   1:  PR[GP1:91,1] = PR[GP1:90,1] + -0.626;
   1:  PR[GP1:91,2] = PR[GP1:90,2] + -44.019;
   1:L PR[91] R[100]mm/sec CNT100;
   1:  PR[GP1:91,1] = PR[GP1:90,1] + 0.841;
   1:L PR[91] R[100]mm/sec CNT100;
   1:  PR[GP1:91,1] = PR[GP1:90,1] + 8.391;
   1:  PR[GP1:91,2] = PR[GP1:90,2] + -44.216;
   1:L PR[91] R[100]mm/sec CNT100;
   1:  PR[GP1:91,1] = PR[GP1:90,1] + 12.992;
   1:  PR[GP1:91,2] = PR[GP1:90,2] + -44.314;
   1:L PR[91] R[100]mm/sec CNT100;
   1:  PR[GP1:91,1] = PR[GP1:90,1] + 15.543;
   1:  PR[GP1:91,2] = PR[GP1:90,2] + -43.998;
   1:L PR[91] R[100]mm/sec CNT100;
   1:  PR[GP1:91,1] = PR[GP1:90,1] + 27.793;
   1:  PR[GP1:91,2] = PR[GP1:90,2] + -39.874;
   1:L PR[91] R[100]mm/sec CNT100;
   1:  PR[GP1:91,1] = PR[GP1:90,1] + 29.749;
   1:  PR[GP1:91,2] = PR[GP1:90,2] + -39.116;
   1:L PR[91] R[100]mm/sec CNT100;
   1:  PR[GP1:91,1] = PR[GP1:90,1] + 40.362;
   1:  PR[GP1:91,2] = PR[GP1:90,2] + -30.633;
   1:L PR[91] R[100]mm/sec CNT100;
   1:  PR[GP1:91,1] = PR[GP1:90,1] + 41.764;
   1:  PR[GP1:91,2] = PR[GP1:90,2] + -29.640;
   1:L PR[91] R[100]mm/sec CNT100;
   1:  PR[GP1:91,1] = PR[GP1:90,1] + 42.961;
   1:  PR[GP1:91,2] = PR[GP1:90,2] + -28.198;
   1:L PR[91] R[100]mm/sec CNT100;
   1:  PR[GP1:91,1] = PR[GP1:90,1] + 49.960;
   1:  PR[GP1:91,2] = PR[GP1:90,2] + -16.511;
   1:L PR[91] R[100]mm/sec CNT100;
   1:  PR[GP1:91,1] = PR[GP1:90,1] + 50.589;
   1:  PR[GP1:91,2] = PR[GP1:90,2] + -15.086;
   1:L PR[91] R[100]mm/sec CNT100;
   1:  PR[GP1:91,1] = PR[GP1:90,1] + 53.075;
   1:  PR[GP1:91,2] = PR[GP1:90,2] + -1.444;
   1:L PR[91] R[100]mm/sec CNT100;
   1:  PR[GP1:91,1] = PR[GP1:90,1] + 53.265;
   1:  PR[GP1:91,2] = PR[GP1:90,2] + -0.085;
   1:L PR[91] R[100]mm/sec CNT100;
   1:  PR[GP1:91,1] = PR[GP1:90,1] + 50.804;
   1:  PR[GP1:91,2] = PR[GP1:90,2] + 13.373;
   1:L PR[91] R[100]mm/sec CNT100;
   1:  PR[GP1:91,1] = PR[GP1:90,1] + 50.584;
   1:  PR[GP1:91,2] = PR[GP1:90,2] + 14.954;
   1:L PR[91] R[100]mm/sec CNT100;
   1:  PR[GP1:91,1] = PR[GP1:90,1] + 49.959;
   1:  PR[GP1:91,2] = PR[GP1:90,2] + 16.368;
   1:L PR[91] R[100]mm/sec CNT100;
   1:  PR[GP1:91,1] = PR[GP1:90,1] + 42.960;
   1:  PR[GP1:91,2] = PR[GP1:90,2] + 28.055;
   1:L PR[91] R[100]mm/sec CNT100;
   1:  PR[GP1:91,1] = PR[GP1:90,1] + 41.751;
   1:  PR[GP1:91,2] = PR[GP1:90,2] + 29.511;
   1:L PR[91] R[100]mm/sec CNT100;
   1:  PR[GP1:91,1] = PR[GP1:90,1] + 31.485;
   1:  PR[GP1:91,2] = PR[GP1:90,2] + 37.748;
   1:L PR[91] R[100]mm/sec CNT100;
   1:  PR[GP1:91,1] = PR[GP1:90,1] + 29.763;
   1:  PR[GP1:91,2] = PR[GP1:90,2] + 38.967;
   1:L PR[91] R[100]mm/sec CNT100;
   1:  PR[GP1:91,1] = PR[GP1:90,1] + 27.791;
   1:  PR[GP1:91,2] = PR[GP1:90,2] + 39.731;
   1:L PR[91] R[100]mm/sec CNT100;
   1:  PR[GP1:91,1] = PR[GP1:90,1] + 15.540;
   1:  PR[GP1:91,2] = PR[GP1:90,2] + 43.855;
   1:L PR[91] R[100]mm/sec CNT100;
   1:  PR[GP1:91,1] = PR[GP1:90,1] + 12.988;
   1:  PR[GP1:91,2] = PR[GP1:90,2] + 44.171;
   1:L PR[91] R[100]mm/sec CNT100;
   1:  PR[GP1:91,1] = PR[GP1:90,1] + 8.403;
   1:  PR[GP1:91,2] = PR[GP1:90,2] + 44.072;
   1:L PR[91] R[100]mm/sec CNT100;
   1:  PR[GP1:91,1] = PR[GP1:90,1] + 0.841;
   1:  PR[GP1:91,2] = PR[GP1:90,2] + 43.875;
   1:L PR[91] R[100]mm/sec CNT100;
   1:  ! -- Layer/Ebene 176 -- !;
   1:  PR[91] = PR[90];
   1:  PR[GP1:91,1] = PR[GP1:90,1] + -0.604;
   1:  PR[GP1:91,2] = PR[GP1:90,2] + 44.034;
   1:  PR[GP1:91,3] = PR[GP1:90,3] + 107.665;
   1:L PR[91] R[100]mm/sec CNT100;
   1:  PR[GP1:91,1] = PR[GP1:90,1] + -7.340;
   1:  PR[GP1:91,2] = PR[GP1:90,2] + 44.210;
   1:L PR[91] R[100]mm/sec CNT100;
   1:  PR[GP1:91,1] = PR[GP1:90,1] + -12.403;
   1:  PR[GP1:91,2] = PR[GP1:90,2] + 44.319;
   1:L PR[91] R[100]mm/sec CNT100;
   1:  PR[GP1:91,1] = PR[GP1:90,1] + -15.228;
   1:  PR[GP1:91,2] = PR[GP1:90,2] + 43.969;
   1:L PR[91] R[100]mm/sec CNT100;
   1:  PR[GP1:91,1] = PR[GP1:90,1] + -27.126;
   1:  PR[GP1:91,2] = PR[GP1:90,2] + 39.965;
   1:L PR[91] R[100]mm/sec CNT100;
   1:  PR[GP1:91,1] = PR[GP1:90,1] + -29.351;
   1:  PR[GP1:91,2] = PR[GP1:90,2] + 39.103;
   1:L PR[91] R[100]mm/sec CNT100;
   1:  PR[GP1:91,1] = PR[GP1:90,1] + -39.660;
   1:  PR[GP1:91,2] = PR[GP1:90,2] + 30.866;
   1:L PR[91] R[100]mm/sec CNT100;
   1:  PR[GP1:91,1] = PR[GP1:90,1] + -41.308;
   1:  PR[GP1:91,2] = PR[GP1:90,2] + 29.699;
   1:L PR[91] R[100]mm/sec CNT100;
   1:  PR[GP1:91,1] = PR[GP1:90,1] + -42.722;
   1:  PR[GP1:91,2] = PR[GP1:90,2] + 27.996;
   1:L PR[91] R[100]mm/sec CNT100;
   1:  PR[GP1:91,1] = PR[GP1:90,1] + -49.520;
   1:  PR[GP1:91,2] = PR[GP1:90,2] + 16.640;
   1:L PR[91] R[100]mm/sec CNT100;
   1:  PR[GP1:91,1] = PR[GP1:90,1] + -50.290;
   1:  PR[GP1:91,2] = PR[GP1:90,2] + 14.895;
   1:L PR[91] R[100]mm/sec CNT100;
   1:  PR[GP1:91,1] = PR[GP1:90,1] + -52.705;
   1:  PR[GP1:91,2] = PR[GP1:90,2] + 1.651;
   1:L PR[91] R[100]mm/sec CNT100;
   1:  PR[GP1:91,1] = PR[GP1:90,1] + -52.943;
   1:  PR[GP1:91,2] = PR[GP1:90,2] + -0.059;
   1:L PR[91] R[100]mm/sec CNT100;
   1:  PR[GP1:91,1] = PR[GP1:90,1] + -50.554;
   1:  PR[GP1:91,2] = PR[GP1:90,2] + -13.124;
   1:L PR[91] R[100]mm/sec CNT100;
   1:  PR[GP1:91,1] = PR[GP1:90,1] + -50.285;
   1:  PR[GP1:91,2] = PR[GP1:90,2] + -15.050;
   1:L PR[91] R[100]mm/sec CNT100;
   1:  PR[GP1:91,1] = PR[GP1:90,1] + -49.520;
   1:  PR[GP1:91,2] = PR[GP1:90,2] + -16.783;
   1:L PR[91] R[100]mm/sec CNT100;
   1:  PR[GP1:91,1] = PR[GP1:90,1] + -42.723;
   1:  PR[GP1:91,2] = PR[GP1:90,2] + -28.138;
   1:L PR[91] R[100]mm/sec CNT100;
   1:  PR[GP1:91,1] = PR[GP1:90,1] + -41.297;
   1:  PR[GP1:91,2] = PR[GP1:90,2] + -29.856;
   1:L PR[91] R[100]mm/sec CNT100;
   1:  PR[GP1:91,1] = PR[GP1:90,1] + -31.328;
   1:  PR[GP1:91,2] = PR[GP1:90,2] + -37.852;
   1:L PR[91] R[100]mm/sec CNT100;
   1:  PR[GP1:91,1] = PR[GP1:90,1] + -29.370;
   1:  PR[GP1:91,2] = PR[GP1:90,2] + -39.239;
   1:L PR[91] R[100]mm/sec CNT100;
   1:  PR[GP1:91,1] = PR[GP1:90,1] + -27.129;
   1:  PR[GP1:91,2] = PR[GP1:90,2] + -40.108;
   1:L PR[91] R[100]mm/sec CNT100;
   1:  PR[GP1:91,1] = PR[GP1:90,1] + -15.231;
   1:  PR[GP1:91,2] = PR[GP1:90,2] + -44.113;
   1:L PR[91] R[100]mm/sec CNT100;
   1:  PR[GP1:91,1] = PR[GP1:90,1] + -12.406;
   1:  PR[GP1:91,2] = PR[GP1:90,2] + -44.463;
   1:L PR[91] R[100]mm/sec CNT100;
   1:  PR[GP1:91,1] = PR[GP1:90,1] + -7.326;
   1:  PR[GP1:91,2] = PR[GP1:90,2] + -44.353;
   1:L PR[91] R[100]mm/sec CNT100;
   1:  PR[GP1:91,1] = PR[GP1:90,1] + -0.604;
   1:  PR[GP1:91,2] = PR[GP1:90,2] + -44.178;
   1:L PR[91] R[100]mm/sec CNT100;
   1:  PR[GP1:91,1] = PR[GP1:90,1] + 0.818;
   1:L PR[91] R[100]mm/sec CNT100;
   1:  PR[GP1:91,1] = PR[GP1:90,1] + 7.540;
   1:  PR[GP1:91,2] = PR[GP1:90,2] + -44.353;
   1:L PR[91] R[100]mm/sec CNT100;
   1:  PR[GP1:91,1] = PR[GP1:90,1] + 12.621;
   1:  PR[GP1:91,2] = PR[GP1:90,2] + -44.462;
   1:L PR[91] R[100]mm/sec CNT100;
   1:  PR[GP1:91,1] = PR[GP1:90,1] + 15.446;
   1:  PR[GP1:91,2] = PR[GP1:90,2] + -44.113;
   1:L PR[91] R[100]mm/sec CNT100;
   1:  PR[GP1:91,1] = PR[GP1:90,1] + 27.343;
   1:  PR[GP1:91,2] = PR[GP1:90,2] + -40.107;
   1:L PR[91] R[100]mm/sec CNT100;
   1:  PR[GP1:91,1] = PR[GP1:90,1] + 29.568;
   1:  PR[GP1:91,2] = PR[GP1:90,2] + -39.245;
   1:L PR[91] R[100]mm/sec CNT100;
   1:  PR[GP1:91,1] = PR[GP1:90,1] + 39.875;
   1:  PR[GP1:91,2] = PR[GP1:90,2] + -31.006;
   1:L PR[91] R[100]mm/sec CNT100;
   1:  PR[GP1:91,1] = PR[GP1:90,1] + 41.523;
   1:  PR[GP1:91,2] = PR[GP1:90,2] + -29.839;
   1:L PR[91] R[100]mm/sec CNT100;
   1:  PR[GP1:91,1] = PR[GP1:90,1] + 42.937;
   1:  PR[GP1:91,2] = PR[GP1:90,2] + -28.136;
   1:L PR[91] R[100]mm/sec CNT100;
   1:  PR[GP1:91,1] = PR[GP1:90,1] + 49.733;
   1:  PR[GP1:91,2] = PR[GP1:90,2] + -16.787;
   1:L PR[91] R[100]mm/sec CNT100;
   1:  PR[GP1:91,1] = PR[GP1:90,1] + 50.504;
   1:  PR[GP1:91,2] = PR[GP1:90,2] + -15.042;
   1:L PR[91] R[100]mm/sec CNT100;
   1:  PR[GP1:91,1] = PR[GP1:90,1] + 52.918;
   1:  PR[GP1:91,2] = PR[GP1:90,2] + -1.795;
   1:L PR[91] R[100]mm/sec CNT100;
   1:  PR[GP1:91,1] = PR[GP1:90,1] + 53.157;
   1:  PR[GP1:91,2] = PR[GP1:90,2] + -0.085;
   1:L PR[91] R[100]mm/sec CNT100;
   1:  PR[GP1:91,1] = PR[GP1:90,1] + 50.767;
   1:  PR[GP1:91,2] = PR[GP1:90,2] + 12.985;
   1:L PR[91] R[100]mm/sec CNT100;
   1:  PR[GP1:91,1] = PR[GP1:90,1] + 50.498;
   1:  PR[GP1:91,2] = PR[GP1:90,2] + 14.911;
   1:L PR[91] R[100]mm/sec CNT100;
   1:  PR[GP1:91,1] = PR[GP1:90,1] + 49.733;
   1:  PR[GP1:91,2] = PR[GP1:90,2] + 16.644;
   1:L PR[91] R[100]mm/sec CNT100;
   1:  PR[GP1:91,1] = PR[GP1:90,1] + 42.936;
   1:  PR[GP1:91,2] = PR[GP1:90,2] + 27.993;
   1:L PR[91] R[100]mm/sec CNT100;
   1:  PR[GP1:91,1] = PR[GP1:90,1] + 41.511;
   1:  PR[GP1:91,2] = PR[GP1:90,2] + 29.710;
   1:L PR[91] R[100]mm/sec CNT100;
   1:  PR[GP1:91,1] = PR[GP1:90,1] + 31.541;
   1:  PR[GP1:91,2] = PR[GP1:90,2] + 37.709;
   1:L PR[91] R[100]mm/sec CNT100;
   1:  PR[GP1:91,1] = PR[GP1:90,1] + 29.583;
   1:  PR[GP1:91,2] = PR[GP1:90,2] + 39.096;
   1:L PR[91] R[100]mm/sec CNT100;
   1:  PR[GP1:91,1] = PR[GP1:90,1] + 27.341;
   1:  PR[GP1:91,2] = PR[GP1:90,2] + 39.964;
   1:L PR[91] R[100]mm/sec CNT100;
   1:  PR[GP1:91,1] = PR[GP1:90,1] + 15.443;
   1:  PR[GP1:91,2] = PR[GP1:90,2] + 43.969;
   1:L PR[91] R[100]mm/sec CNT100;
   1:  PR[GP1:91,1] = PR[GP1:90,1] + 12.618;
   1:  PR[GP1:91,2] = PR[GP1:90,2] + 44.319;
   1:L PR[91] R[100]mm/sec CNT100;
   1:  PR[GP1:91,1] = PR[GP1:90,1] + 7.554;
   1:  PR[GP1:91,2] = PR[GP1:90,2] + 44.210;
   1:L PR[91] R[100]mm/sec CNT100;
   1:  PR[GP1:91,1] = PR[GP1:90,1] + 0.818;
   1:  PR[GP1:91,2] = PR[GP1:90,2] + 44.034;
   1:L PR[91] R[100]mm/sec CNT100;
   1:  ! -- Layer/Ebene 177 -- !;
   1:  PR[91] = PR[90];
   1:  PR[GP1:91,1] = PR[GP1:90,1] + -0.581;
   1:  PR[GP1:91,2] = PR[GP1:90,2] + 44.194;
   1:  PR[GP1:91,3] = PR[GP1:90,3] + 108.275;
   1:L PR[91] R[100]mm/sec CNT100;
   1:  PR[GP1:91,1] = PR[GP1:90,1] + -6.491;
   1:  PR[GP1:91,2] = PR[GP1:90,2] + 44.348;
   1:L PR[91] R[100]mm/sec CNT100;
   1:  PR[GP1:91,1] = PR[GP1:90,1] + -12.033;
   1:  PR[GP1:91,2] = PR[GP1:90,2] + 44.467;
   1:L PR[91] R[100]mm/sec CNT100;
   1:  PR[GP1:91,1] = PR[GP1:90,1] + -15.132;
   1:  PR[GP1:91,2] = PR[GP1:90,2] + 44.083;
   1:L PR[91] R[100]mm/sec CNT100;
   1:  PR[GP1:91,1] = PR[GP1:90,1] + -26.676;
   1:  PR[GP1:91,2] = PR[GP1:90,2] + 40.198;
   1:L PR[91] R[100]mm/sec CNT100;
   1:  PR[GP1:91,1] = PR[GP1:90,1] + -29.171;
   1:  PR[GP1:91,2] = PR[GP1:90,2] + 39.231;
   1:L PR[91] R[100]mm/sec CNT100;
   1:  PR[GP1:91,1] = PR[GP1:90,1] + -39.173;
   1:  PR[GP1:91,2] = PR[GP1:90,2] + 31.240;
   1:L PR[91] R[100]mm/sec CNT100;
   1:  PR[GP1:91,1] = PR[GP1:90,1] + -41.068;
   1:  PR[GP1:91,2] = PR[GP1:90,2] + 29.898;
   1:L PR[91] R[100]mm/sec CNT100;
   1:  PR[GP1:91,1] = PR[GP1:90,1] + -42.698;
   1:  PR[GP1:91,2] = PR[GP1:90,2] + 27.934;
   1:L PR[91] R[100]mm/sec CNT100;
   1:  PR[GP1:91,1] = PR[GP1:90,1] + -49.294;
   1:  PR[GP1:91,2] = PR[GP1:90,2] + 16.916;
   1:L PR[91] R[100]mm/sec CNT100;
   1:  PR[GP1:91,1] = PR[GP1:90,1] + -50.205;
   1:  PR[GP1:91,2] = PR[GP1:90,2] + 14.852;
   1:L PR[91] R[100]mm/sec CNT100;
   1:  PR[GP1:91,1] = PR[GP1:90,1] + -52.548;
   1:  PR[GP1:91,2] = PR[GP1:90,2] + 2.002;
   1:L PR[91] R[100]mm/sec CNT100;
   1:  PR[GP1:91,1] = PR[GP1:90,1] + -52.835;
   1:  PR[GP1:91,2] = PR[GP1:90,2] + -0.059;
   1:L PR[91] R[100]mm/sec CNT100;
   1:  PR[GP1:91,1] = PR[GP1:90,1] + -50.517;
   1:  PR[GP1:91,2] = PR[GP1:90,2] + -12.735;
   1:L PR[91] R[100]mm/sec CNT100;
   1:  PR[GP1:91,1] = PR[GP1:90,1] + -50.200;
   1:  PR[GP1:91,2] = PR[GP1:90,2] + -15.007;
   1:L PR[91] R[100]mm/sec CNT100;
   1:  PR[GP1:91,1] = PR[GP1:90,1] + -49.294;
   1:  PR[GP1:91,2] = PR[GP1:90,2] + -17.059;
   1:L PR[91] R[100]mm/sec CNT100;
   1:  PR[GP1:91,1] = PR[GP1:90,1] + -42.699;
   1:  PR[GP1:91,2] = PR[GP1:90,2] + -28.076;
   1:L PR[91] R[100]mm/sec CNT100;
   1:  PR[GP1:91,1] = PR[GP1:90,1] + -41.057;
   1:  PR[GP1:91,2] = PR[GP1:90,2] + -30.055;
   1:L PR[91] R[100]mm/sec CNT100;
   1:  PR[GP1:91,1] = PR[GP1:90,1] + -31.384;
   1:  PR[GP1:91,2] = PR[GP1:90,2] + -37.813;
   1:L PR[91] R[100]mm/sec CNT100;
   1:  PR[GP1:91,1] = PR[GP1:90,1] + -29.190;
   1:  PR[GP1:91,2] = PR[GP1:90,2] + -39.367;
   1:L PR[91] R[100]mm/sec CNT100;
   1:  PR[GP1:91,1] = PR[GP1:90,1] + -26.678;
   1:  PR[GP1:91,2] = PR[GP1:90,2] + -40.341;
   1:L PR[91] R[100]mm/sec CNT100;
   1:  PR[GP1:91,1] = PR[GP1:90,1] + -15.135;
   1:  PR[GP1:91,2] = PR[GP1:90,2] + -44.227;
   1:L PR[91] R[100]mm/sec CNT100;
   1:  PR[GP1:91,1] = PR[GP1:90,1] + -12.036;
   1:  PR[GP1:91,2] = PR[GP1:90,2] + -44.611;
   1:L PR[91] R[100]mm/sec CNT100;
   1:  PR[GP1:91,1] = PR[GP1:90,1] + -6.476;
   1:  PR[GP1:91,2] = PR[GP1:90,2] + -44.491;
   1:L PR[91] R[100]mm/sec CNT100;
   1:  PR[GP1:91,1] = PR[GP1:90,1] + -0.581;
   1:  PR[GP1:91,2] = PR[GP1:90,2] + -44.338;
   1:L PR[91] R[100]mm/sec CNT100;
   1:  PR[GP1:91,1] = PR[GP1:90,1] + 0.795;
   1:L PR[91] R[100]mm/sec CNT100;
   1:  PR[GP1:91,1] = PR[GP1:90,1] + 6.690;
   1:  PR[GP1:91,2] = PR[GP1:90,2] + -44.491;
   1:L PR[91] R[100]mm/sec CNT100;
   1:  PR[GP1:91,1] = PR[GP1:90,1] + 12.250;
   1:  PR[GP1:91,2] = PR[GP1:90,2] + -44.610;
   1:L PR[91] R[100]mm/sec CNT100;
   1:  PR[GP1:91,1] = PR[GP1:90,1] + 15.349;
   1:  PR[GP1:91,2] = PR[GP1:90,2] + -44.227;
   1:L PR[91] R[100]mm/sec CNT100;
   1:  PR[GP1:91,1] = PR[GP1:90,1] + 26.893;
   1:  PR[GP1:91,2] = PR[GP1:90,2] + -40.340;
   1:L PR[91] R[100]mm/sec CNT100;
   1:  PR[GP1:91,1] = PR[GP1:90,1] + 29.388;
   1:  PR[GP1:91,2] = PR[GP1:90,2] + -39.373;
   1:L PR[91] R[100]mm/sec CNT100;
   1:  PR[GP1:91,1] = PR[GP1:90,1] + 39.388;
   1:  PR[GP1:91,2] = PR[GP1:90,2] + -31.380;
   1:L PR[91] R[100]mm/sec CNT100;
   1:  PR[GP1:91,1] = PR[GP1:90,1] + 41.283;
   1:  PR[GP1:91,2] = PR[GP1:90,2] + -30.038;
   1:L PR[91] R[100]mm/sec CNT100;
   1:  PR[GP1:91,1] = PR[GP1:90,1] + 42.914;
   1:  PR[GP1:91,2] = PR[GP1:90,2] + -28.074;
   1:L PR[91] R[100]mm/sec CNT100;
   1:  PR[GP1:91,1] = PR[GP1:90,1] + 49.508;
   1:  PR[GP1:91,2] = PR[GP1:90,2] + -17.063;
   1:L PR[91] R[100]mm/sec CNT100;
   1:  PR[GP1:91,1] = PR[GP1:90,1] + 50.419;
   1:  PR[GP1:91,2] = PR[GP1:90,2] + -14.999;
   1:L PR[91] R[100]mm/sec CNT100;
   1:  PR[GP1:91,1] = PR[GP1:90,1] + 52.761;
   1:  PR[GP1:91,2] = PR[GP1:90,2] + -2.146;
   1:L PR[91] R[100]mm/sec CNT100;
   1:  PR[GP1:91,1] = PR[GP1:90,1] + 53.048;
   1:  PR[GP1:91,2] = PR[GP1:90,2] + -0.085;
   1:L PR[91] R[100]mm/sec CNT100;
   1:  PR[GP1:91,1] = PR[GP1:90,1] + 50.730;
   1:  PR[GP1:91,2] = PR[GP1:90,2] + 12.596;
   1:L PR[91] R[100]mm/sec CNT100;
   1:  PR[GP1:91,1] = PR[GP1:90,1] + 50.413;
   1:  PR[GP1:91,2] = PR[GP1:90,2] + 14.867;
   1:L PR[91] R[100]mm/sec CNT100;
   1:  PR[GP1:91,1] = PR[GP1:90,1] + 49.507;
   1:  PR[GP1:91,2] = PR[GP1:90,2] + 16.919;
   1:L PR[91] R[100]mm/sec CNT100;
   1:  PR[GP1:91,1] = PR[GP1:90,1] + 42.912;
   1:  PR[GP1:91,2] = PR[GP1:90,2] + 27.931;
   1:L PR[91] R[100]mm/sec CNT100;
   1:  PR[GP1:91,1] = PR[GP1:90,1] + 41.270;
   1:  PR[GP1:91,2] = PR[GP1:90,2] + 29.909;
   1:L PR[91] R[100]mm/sec CNT100;
   1:  PR[GP1:91,1] = PR[GP1:90,1] + 31.597;
   1:  PR[GP1:91,2] = PR[GP1:90,2] + 37.670;
   1:L PR[91] R[100]mm/sec CNT100;
   1:  PR[GP1:91,1] = PR[GP1:90,1] + 29.402;
   1:  PR[GP1:91,2] = PR[GP1:90,2] + 39.224;
   1:L PR[91] R[100]mm/sec CNT100;
   1:  PR[GP1:91,1] = PR[GP1:90,1] + 26.890;
   1:  PR[GP1:91,2] = PR[GP1:90,2] + 40.198;
   1:L PR[91] R[100]mm/sec CNT100;
   1:  PR[GP1:91,1] = PR[GP1:90,1] + 15.346;
   1:  PR[GP1:91,2] = PR[GP1:90,2] + 44.083;
   1:L PR[91] R[100]mm/sec CNT100;
   1:  PR[GP1:91,1] = PR[GP1:90,1] + 12.247;
   1:  PR[GP1:91,2] = PR[GP1:90,2] + 44.467;
   1:L PR[91] R[100]mm/sec CNT100;
   1:  PR[GP1:91,1] = PR[GP1:90,1] + 6.705;
   1:  PR[GP1:91,2] = PR[GP1:90,2] + 44.348;
   1:L PR[91] R[100]mm/sec CNT100;
   1:  PR[GP1:91,1] = PR[GP1:90,1] + 0.795;
   1:  PR[GP1:91,2] = PR[GP1:90,2] + 44.194;
   1:L PR[91] R[100]mm/sec CNT100;
   1:  ! -- Layer/Ebene 178 -- !;
   1:  PR[91] = PR[90];
   1:  PR[GP1:91,1] = PR[GP1:90,1] + -0.559;
   1:  PR[GP1:91,2] = PR[GP1:90,2] + 44.353;
   1:  PR[GP1:91,3] = PR[GP1:90,3] + 108.885;
   1:L PR[91] R[100]mm/sec CNT100;
   1:  PR[GP1:91,1] = PR[GP1:90,1] + -5.642;
   1:  PR[GP1:91,2] = PR[GP1:90,2] + 44.486;
   1:L PR[91] R[100]mm/sec CNT100;
   1:  PR[GP1:91,1] = PR[GP1:90,1] + -11.662;
   1:  PR[GP1:91,2] = PR[GP1:90,2] + 44.615;
   1:L PR[91] R[100]mm/sec CNT100;
   1:  PR[GP1:91,1] = PR[GP1:90,1] + -15.035;
   1:  PR[GP1:91,2] = PR[GP1:90,2] + 44.197;
   1:L PR[91] R[100]mm/sec CNT100;
   1:  PR[GP1:91,1] = PR[GP1:90,1] + -26.226;
   1:  PR[GP1:91,2] = PR[GP1:90,2] + 40.431;
   1:L PR[91] R[100]mm/sec CNT100;
   1:  PR[GP1:91,1] = PR[GP1:90,1] + -28.991;
   1:  PR[GP1:91,2] = PR[GP1:90,2] + 39.359;
   1:L PR[91] R[100]mm/sec CNT100;
   1:  PR[GP1:91,1] = PR[GP1:90,1] + -38.686;
   1:  PR[GP1:91,2] = PR[GP1:90,2] + 31.613;
   1:L PR[91] R[100]mm/sec CNT100;
   1:  PR[GP1:91,1] = PR[GP1:90,1] + -40.827;
   1:  PR[GP1:91,2] = PR[GP1:90,2] + 30.097;
   1:L PR[91] R[100]mm/sec CNT100;
   1:  PR[GP1:91,1] = PR[GP1:90,1] + -42.675;
   1:  PR[GP1:91,2] = PR[GP1:90,2] + 27.872;
   1:L PR[91] R[100]mm/sec CNT100;
   1:  PR[GP1:91,1] = PR[GP1:90,1] + -49.068;
   1:  PR[GP1:91,2] = PR[GP1:90,2] + 17.191;
   1:L PR[91] R[100]mm/sec CNT100;
   1:  PR[GP1:91,1] = PR[GP1:90,1] + -50.120;
   1:  PR[GP1:91,2] = PR[GP1:90,2] + 14.809;
   1:L PR[91] R[100]mm/sec CNT100;
   1:  PR[GP1:91,1] = PR[GP1:90,1] + -52.391;
   1:  PR[GP1:91,2] = PR[GP1:90,2] + 2.352;
   1:L PR[91] R[100]mm/sec CNT100;
   1:  PR[GP1:91,1] = PR[GP1:90,1] + -52.727;
   1:  PR[GP1:91,2] = PR[GP1:90,2] + -0.059;
   1:L PR[91] R[100]mm/sec CNT100;
   1:  PR[GP1:91,1] = PR[GP1:90,1] + -50.480;
   1:  PR[GP1:91,2] = PR[GP1:90,2] + -12.347;
   1:L PR[91] R[100]mm/sec CNT100;
   1:  PR[GP1:91,1] = PR[GP1:90,1] + -50.115;
   1:  PR[GP1:91,2] = PR[GP1:90,2] + -14.963;
   1:L PR[91] R[100]mm/sec CNT100;
   1:  PR[GP1:91,1] = PR[GP1:90,1] + -49.068;
   1:  PR[GP1:91,2] = PR[GP1:90,2] + -17.335;
   1:L PR[91] R[100]mm/sec CNT100;
   1:  PR[GP1:91,1] = PR[GP1:90,1] + -42.676;
   1:  PR[GP1:91,2] = PR[GP1:90,2] + -28.014;
   1:L PR[91] R[100]mm/sec CNT100;
   1:  PR[GP1:91,1] = PR[GP1:90,1] + -40.817;
   1:  PR[GP1:91,2] = PR[GP1:90,2] + -30.254;
   1:L PR[91] R[100]mm/sec CNT100;
   1:  PR[GP1:91,1] = PR[GP1:90,1] + -31.440;
   1:  PR[GP1:91,2] = PR[GP1:90,2] + -37.774;
   1:L PR[91] R[100]mm/sec CNT100;
   1:  PR[GP1:91,1] = PR[GP1:90,1] + -29.009;
   1:  PR[GP1:91,2] = PR[GP1:90,2] + -39.496;
   1:L PR[91] R[100]mm/sec CNT100;
   1:  PR[GP1:91,1] = PR[GP1:90,1] + -26.228;
   1:  PR[GP1:91,2] = PR[GP1:90,2] + -40.574;
   1:L PR[91] R[100]mm/sec CNT100;
   1:  PR[GP1:91,1] = PR[GP1:90,1] + -15.038;
   1:  PR[GP1:91,2] = PR[GP1:90,2] + -44.341;
   1:L PR[91] R[100]mm/sec CNT100;
   1:  PR[GP1:91,1] = PR[GP1:90,1] + -11.665;
   1:  PR[GP1:91,2] = PR[GP1:90,2] + -44.759;
   1:L PR[91] R[100]mm/sec CNT100;
   1:  PR[GP1:91,1] = PR[GP1:90,1] + -5.625;
   1:  PR[GP1:91,2] = PR[GP1:90,2] + -44.629;
   1:L PR[91] R[100]mm/sec CNT100;
   1:  PR[GP1:91,1] = PR[GP1:90,1] + -0.559;
   1:  PR[GP1:91,2] = PR[GP1:90,2] + -44.497;
   1:L PR[91] R[100]mm/sec CNT100;
   1:  PR[GP1:91,1] = PR[GP1:90,1] + 0.772;
   1:L PR[91] R[100]mm/sec CNT100;
   1:  PR[GP1:91,1] = PR[GP1:90,1] + 5.839;
   1:  PR[GP1:91,2] = PR[GP1:90,2] + -44.629;
   1:L PR[91] R[100]mm/sec CNT100;
   1:  PR[GP1:91,1] = PR[GP1:90,1] + 11.879;
   1:  PR[GP1:91,2] = PR[GP1:90,2] + -44.759;
   1:L PR[91] R[100]mm/sec CNT100;
   1:  PR[GP1:91,1] = PR[GP1:90,1] + 15.252;
   1:  PR[GP1:91,2] = PR[GP1:90,2] + -44.341;
   1:L PR[91] R[100]mm/sec CNT100;
   1:  PR[GP1:91,1] = PR[GP1:90,1] + 26.442;
   1:  PR[GP1:91,2] = PR[GP1:90,2] + -40.573;
   1:L PR[91] R[100]mm/sec CNT100;
   1:  PR[GP1:91,1] = PR[GP1:90,1] + 29.207;
   1:  PR[GP1:91,2] = PR[GP1:90,2] + -39.502;
   1:L PR[91] R[100]mm/sec CNT100;
   1:  PR[GP1:91,1] = PR[GP1:90,1] + 38.901;
   1:  PR[GP1:91,2] = PR[GP1:90,2] + -31.753;
   1:L PR[91] R[100]mm/sec CNT100;
   1:  PR[GP1:91,1] = PR[GP1:90,1] + 41.043;
   1:  PR[GP1:91,2] = PR[GP1:90,2] + -30.237;
   1:L PR[91] R[100]mm/sec CNT100;
   1:  PR[GP1:91,1] = PR[GP1:90,1] + 42.890;
   1:  PR[GP1:91,2] = PR[GP1:90,2] + -28.012;
   1:L PR[91] R[100]mm/sec CNT100;
   1:  PR[GP1:91,1] = PR[GP1:90,1] + 49.282;
   1:  PR[GP1:91,2] = PR[GP1:90,2] + -17.338;
   1:L PR[91] R[100]mm/sec CNT100;
   1:  PR[GP1:91,1] = PR[GP1:90,1] + 50.333;
   1:  PR[GP1:91,2] = PR[GP1:90,2] + -14.956;
   1:L PR[91] R[100]mm/sec CNT100;
   1:  PR[GP1:91,1] = PR[GP1:90,1] + 52.604;
   1:  PR[GP1:91,2] = PR[GP1:90,2] + -2.496;
   1:L PR[91] R[100]mm/sec CNT100;
   1:  PR[GP1:91,1] = PR[GP1:90,1] + 52.940;
   1:  PR[GP1:91,2] = PR[GP1:90,2] + -0.085;
   1:L PR[91] R[100]mm/sec CNT100;
   1:  PR[GP1:91,1] = PR[GP1:90,1] + 50.693;
   1:  PR[GP1:91,2] = PR[GP1:90,2] + 12.207;
   1:L PR[91] R[100]mm/sec CNT100;
   1:  PR[GP1:91,1] = PR[GP1:90,1] + 50.328;
   1:  PR[GP1:91,2] = PR[GP1:90,2] + 14.824;
   1:L PR[91] R[100]mm/sec CNT100;
   1:  PR[GP1:91,1] = PR[GP1:90,1] + 49.281;
   1:  PR[GP1:91,2] = PR[GP1:90,2] + 17.195;
   1:L PR[91] R[100]mm/sec CNT100;
   1:  PR[GP1:91,1] = PR[GP1:90,1] + 42.889;
   1:  PR[GP1:91,2] = PR[GP1:90,2] + 27.869;
   1:L PR[91] R[100]mm/sec CNT100;
   1:  PR[GP1:91,1] = PR[GP1:90,1] + 41.030;
   1:  PR[GP1:91,2] = PR[GP1:90,2] + 30.108;
   1:L PR[91] R[100]mm/sec CNT100;
   1:  PR[GP1:91,1] = PR[GP1:90,1] + 31.653;
   1:  PR[GP1:91,2] = PR[GP1:90,2] + 37.631;
   1:L PR[91] R[100]mm/sec CNT100;
   1:  PR[GP1:91,1] = PR[GP1:90,1] + 29.222;
   1:  PR[GP1:91,2] = PR[GP1:90,2] + 39.353;
   1:L PR[91] R[100]mm/sec CNT100;
   1:  PR[GP1:91,1] = PR[GP1:90,1] + 26.440;
   1:  PR[GP1:91,2] = PR[GP1:90,2] + 40.431;
   1:L PR[91] R[100]mm/sec CNT100;
   1:  PR[GP1:91,1] = PR[GP1:90,1] + 15.250;
   1:  PR[GP1:91,2] = PR[GP1:90,2] + 44.197;
   1:L PR[91] R[100]mm/sec CNT100;
   1:  PR[GP1:91,1] = PR[GP1:90,1] + 11.876;
   1:  PR[GP1:91,2] = PR[GP1:90,2] + 44.615;
   1:L PR[91] R[100]mm/sec CNT100;
   1:  PR[GP1:91,1] = PR[GP1:90,1] + 5.857;
   1:  PR[GP1:91,2] = PR[GP1:90,2] + 44.485;
   1:L PR[91] R[100]mm/sec CNT100;
   1:  PR[GP1:91,1] = PR[GP1:90,1] + 0.772;
   1:  PR[GP1:91,2] = PR[GP1:90,2] + 44.353;
   1:L PR[91] R[100]mm/sec CNT100;
   1:  ! -- Layer/Ebene 179 -- !;
   1:  PR[91] = PR[90];
   1:  PR[GP1:91,1] = PR[GP1:90,1] + -0.536;
   1:  PR[GP1:91,2] = PR[GP1:90,2] + 44.512;
   1:  PR[GP1:91,3] = PR[GP1:90,3] + 109.495;
   1:L PR[91] R[100]mm/sec CNT100;
   1:  PR[GP1:91,1] = PR[GP1:90,1] + -4.794;
   1:  PR[GP1:91,2] = PR[GP1:90,2] + 44.623;
   1:L PR[91] R[100]mm/sec CNT100;
   1:  PR[GP1:91,1] = PR[GP1:90,1] + -11.291;
   1:  PR[GP1:91,2] = PR[GP1:90,2] + 44.763;
   1:L PR[91] R[100]mm/sec CNT100;
   1:  PR[GP1:91,1] = PR[GP1:90,1] + -14.938;
   1:  PR[GP1:91,2] = PR[GP1:90,2] + 44.311;
   1:L PR[91] R[100]mm/sec CNT100;
   1:  PR[GP1:91,1] = PR[GP1:90,1] + -25.775;
   1:  PR[GP1:91,2] = PR[GP1:90,2] + 40.664;
   1:L PR[91] R[100]mm/sec CNT100;
   1:  PR[GP1:91,1] = PR[GP1:90,1] + -28.811;
   1:  PR[GP1:91,2] = PR[GP1:90,2] + 39.488;
   1:L PR[91] R[100]mm/sec CNT100;
   1:  PR[GP1:91,1] = PR[GP1:90,1] + -38.200;
   1:  PR[GP1:91,2] = PR[GP1:90,2] + 31.986;
   1:L PR[91] R[100]mm/sec CNT100;
   1:  PR[GP1:91,1] = PR[GP1:90,1] + -40.587;
   1:  PR[GP1:91,2] = PR[GP1:90,2] + 30.296;
   1:L PR[91] R[100]mm/sec CNT100;
   1:  PR[GP1:91,1] = PR[GP1:90,1] + -42.651;
   1:  PR[GP1:91,2] = PR[GP1:90,2] + 27.810;
   1:L PR[91] R[100]mm/sec CNT100;
   1:  PR[GP1:91,1] = PR[GP1:90,1] + -48.842;
   1:  PR[GP1:91,2] = PR[GP1:90,2] + 17.467;
   1:L PR[91] R[100]mm/sec CNT100;
   1:  PR[GP1:91,1] = PR[GP1:90,1] + -50.034;
   1:  PR[GP1:91,2] = PR[GP1:90,2] + 14.765;
   1:L PR[91] R[100]mm/sec CNT100;
   1:  PR[GP1:91,1] = PR[GP1:90,1] + -52.234;
   1:  PR[GP1:91,2] = PR[GP1:90,2] + 2.703;
   1:L PR[91] R[100]mm/sec CNT100;
   1:  PR[GP1:91,1] = PR[GP1:90,1] + -52.619;
   1:  PR[GP1:91,2] = PR[GP1:90,2] + -0.059;
   1:L PR[91] R[100]mm/sec CNT100;
   1:  PR[GP1:91,1] = PR[GP1:90,1] + -50.443;
   1:  PR[GP1:91,2] = PR[GP1:90,2] + -11.958;
   1:L PR[91] R[100]mm/sec CNT100;
   1:  PR[GP1:91,1] = PR[GP1:90,1] + -50.030;
   1:  PR[GP1:91,2] = PR[GP1:90,2] + -14.920;
   1:L PR[91] R[100]mm/sec CNT100;
   1:  PR[GP1:91,1] = PR[GP1:90,1] + -48.842;
   1:  PR[GP1:91,2] = PR[GP1:90,2] + -17.610;
   1:L PR[91] R[100]mm/sec CNT100;
   1:  PR[GP1:91,1] = PR[GP1:90,1] + -42.652;
   1:  PR[GP1:91,2] = PR[GP1:90,2] + -27.953;
   1:L PR[91] R[100]mm/sec CNT100;
   1:  PR[GP1:91,1] = PR[GP1:90,1] + -40.576;
   1:  PR[GP1:91,2] = PR[GP1:90,2] + -30.453;
   1:L PR[91] R[100]mm/sec CNT100;
   1:  PR[GP1:91,1] = PR[GP1:90,1] + -31.496;
   1:  PR[GP1:91,2] = PR[GP1:90,2] + -37.736;
   1:L PR[91] R[100]mm/sec CNT100;
   1:  PR[GP1:91,1] = PR[GP1:90,1] + -28.829;
   1:  PR[GP1:91,2] = PR[GP1:90,2] + -39.624;
   1:L PR[91] R[100]mm/sec CNT100;
   1:  PR[GP1:91,1] = PR[GP1:90,1] + -25.777;
   1:  PR[GP1:91,2] = PR[GP1:90,2] + -40.807;
   1:L PR[91] R[100]mm/sec CNT100;
   1:  PR[GP1:91,1] = PR[GP1:90,1] + -14.941;
   1:  PR[GP1:91,2] = PR[GP1:90,2] + -44.455;
   1:L PR[91] R[100]mm/sec CNT100;
   1:  PR[GP1:91,1] = PR[GP1:90,1] + -11.294;
   1:  PR[GP1:91,2] = PR[GP1:90,2] + -44.907;
   1:L PR[91] R[100]mm/sec CNT100;
   1:  PR[GP1:91,1] = PR[GP1:90,1] + -4.775;
   1:  PR[GP1:91,2] = PR[GP1:90,2] + -44.767;
   1:L PR[91] R[100]mm/sec CNT100;
   1:  PR[GP1:91,1] = PR[GP1:90,1] + -0.536;
   1:  PR[GP1:91,2] = PR[GP1:90,2] + -44.656;
   1:L PR[91] R[100]mm/sec CNT100;
   1:  PR[GP1:91,1] = PR[GP1:90,1] + 0.750;
   1:L PR[91] R[100]mm/sec CNT100;
   1:  PR[GP1:91,1] = PR[GP1:90,1] + 4.989;
   1:  PR[GP1:91,2] = PR[GP1:90,2] + -44.767;
   1:L PR[91] R[100]mm/sec CNT100;
   1:  PR[GP1:91,1] = PR[GP1:90,1] + 11.508;
   1:  PR[GP1:91,2] = PR[GP1:90,2] + -44.907;
   1:L PR[91] R[100]mm/sec CNT100;
   1:  PR[GP1:91,1] = PR[GP1:90,1] + 15.156;
   1:  PR[GP1:91,2] = PR[GP1:90,2] + -44.455;
   1:L PR[91] R[100]mm/sec CNT100;
   1:  PR[GP1:91,1] = PR[GP1:90,1] + 25.992;
   1:  PR[GP1:91,2] = PR[GP1:90,2] + -40.807;
   1:L PR[91] R[100]mm/sec CNT100;
   1:  PR[GP1:91,1] = PR[GP1:90,1] + 29.027;
   1:  PR[GP1:91,2] = PR[GP1:90,2] + -39.631;
   1:L PR[91] R[100]mm/sec CNT100;
   1:  PR[GP1:91,1] = PR[GP1:90,1] + 38.415;
   1:  PR[GP1:91,2] = PR[GP1:90,2] + -32.127;
   1:L PR[91] R[100]mm/sec CNT100;
   1:  PR[GP1:91,1] = PR[GP1:90,1] + 40.802;
   1:  PR[GP1:91,2] = PR[GP1:90,2] + -30.436;
   1:L PR[91] R[100]mm/sec CNT100;
   1:  PR[GP1:91,1] = PR[GP1:90,1] + 42.866;
   1:  PR[GP1:91,2] = PR[GP1:90,2] + -27.950;
   1:L PR[91] R[100]mm/sec CNT100;
   1:  PR[GP1:91,1] = PR[GP1:90,1] + 49.055;
   1:  PR[GP1:91,2] = PR[GP1:90,2] + -17.614;
   1:L PR[91] R[100]mm/sec CNT100;
   1:  PR[GP1:91,1] = PR[GP1:90,1] + 50.248;
   1:  PR[GP1:91,2] = PR[GP1:90,2] + -14.912;
   1:L PR[91] R[100]mm/sec CNT100;
   1:  PR[GP1:91,1] = PR[GP1:90,1] + 52.447;
   1:  PR[GP1:91,2] = PR[GP1:90,2] + -2.847;
   1:L PR[91] R[100]mm/sec CNT100;
   1:  PR[GP1:91,1] = PR[GP1:90,1] + 52.832;
   1:  PR[GP1:91,2] = PR[GP1:90,2] + -0.085;
   1:L PR[91] R[100]mm/sec CNT100;
   1:  PR[GP1:91,1] = PR[GP1:90,1] + 50.656;
   1:  PR[GP1:91,2] = PR[GP1:90,2] + 11.819;
   1:L PR[91] R[100]mm/sec CNT100;
   1:  PR[GP1:91,1] = PR[GP1:90,1] + 50.243;
   1:  PR[GP1:91,2] = PR[GP1:90,2] + 14.781;
   1:L PR[91] R[100]mm/sec CNT100;
   1:  PR[GP1:91,1] = PR[GP1:90,1] + 49.055;
   1:  PR[GP1:91,2] = PR[GP1:90,2] + 17.471;
   1:L PR[91] R[100]mm/sec CNT100;
   1:  PR[GP1:91,1] = PR[GP1:90,1] + 42.865;
   1:  PR[GP1:91,2] = PR[GP1:90,2] + 27.807;
   1:L PR[91] R[100]mm/sec CNT100;
   1:  PR[GP1:91,1] = PR[GP1:90,1] + 40.789;
   1:  PR[GP1:91,2] = PR[GP1:90,2] + 30.307;
   1:L PR[91] R[100]mm/sec CNT100;
   1:  PR[GP1:91,1] = PR[GP1:90,1] + 31.709;
   1:  PR[GP1:91,2] = PR[GP1:90,2] + 37.592;
   1:L PR[91] R[100]mm/sec CNT100;
   1:  PR[GP1:91,1] = PR[GP1:90,1] + 29.042;
   1:  PR[GP1:91,2] = PR[GP1:90,2] + 39.481;
   1:L PR[91] R[100]mm/sec CNT100;
   1:  PR[GP1:91,1] = PR[GP1:90,1] + 25.990;
   1:  PR[GP1:91,2] = PR[GP1:90,2] + 40.664;
   1:L PR[91] R[100]mm/sec CNT100;
   1:  PR[GP1:91,1] = PR[GP1:90,1] + 15.153;
   1:  PR[GP1:91,2] = PR[GP1:90,2] + 44.311;
   1:L PR[91] R[100]mm/sec CNT100;
   1:  PR[GP1:91,1] = PR[GP1:90,1] + 11.505;
   1:  PR[GP1:91,2] = PR[GP1:90,2] + 44.763;
   1:L PR[91] R[100]mm/sec CNT100;
   1:  PR[GP1:91,1] = PR[GP1:90,1] + 5.008;
   1:  PR[GP1:91,2] = PR[GP1:90,2] + 44.623;
   1:L PR[91] R[100]mm/sec CNT100;
   1:  PR[GP1:91,1] = PR[GP1:90,1] + 0.750;
   1:  PR[GP1:91,2] = PR[GP1:90,2] + 44.512;
   1:L PR[91] R[100]mm/sec CNT100;
   1:  ! -- Layer/Ebene 180 -- !;
   1:  PR[91] = PR[90];
   1:  PR[GP1:91,1] = PR[GP1:90,1] + -0.513;
   1:  PR[GP1:91,2] = PR[GP1:90,2] + 44.671;
   1:  PR[GP1:91,3] = PR[GP1:90,3] + 110.105;
   1:L PR[91] R[100]mm/sec CNT100;
   1:  PR[GP1:91,1] = PR[GP1:90,1] + -3.945;
   1:  PR[GP1:91,2] = PR[GP1:90,2] + 44.761;
   1:L PR[91] R[100]mm/sec CNT100;
   1:  PR[GP1:91,1] = PR[GP1:90,1] + -10.921;
   1:  PR[GP1:91,2] = PR[GP1:90,2] + 44.911;
   1:L PR[91] R[100]mm/sec CNT100;
   1:  PR[GP1:91,1] = PR[GP1:90,1] + -14.842;
   1:  PR[GP1:91,2] = PR[GP1:90,2] + 44.425;
   1:L PR[91] R[100]mm/sec CNT100;
   1:  PR[GP1:91,1] = PR[GP1:90,1] + -25.325;
   1:  PR[GP1:91,2] = PR[GP1:90,2] + 40.897;
   1:L PR[91] R[100]mm/sec CNT100;
   1:  PR[GP1:91,1] = PR[GP1:90,1] + -28.630;
   1:  PR[GP1:91,2] = PR[GP1:90,2] + 39.616;
   1:L PR[91] R[100]mm/sec CNT100;
   1:  PR[GP1:91,1] = PR[GP1:90,1] + -37.713;
   1:  PR[GP1:91,2] = PR[GP1:90,2] + 32.359;
   1:L PR[91] R[100]mm/sec CNT100;
   1:  PR[GP1:91,1] = PR[GP1:90,1] + -40.346;
   1:  PR[GP1:91,2] = PR[GP1:90,2] + 30.495;
   1:L PR[91] R[100]mm/sec CNT100;
   1:  PR[GP1:91,1] = PR[GP1:90,1] + -42.627;
   1:  PR[GP1:91,2] = PR[GP1:90,2] + 27.748;
   1:L PR[91] R[100]mm/sec CNT100;
   1:  PR[GP1:91,1] = PR[GP1:90,1] + -48.616;
   1:  PR[GP1:91,2] = PR[GP1:90,2] + 17.743;
   1:L PR[91] R[100]mm/sec CNT100;
   1:  PR[GP1:91,1] = PR[GP1:90,1] + -49.949;
   1:  PR[GP1:91,2] = PR[GP1:90,2] + 14.722;
   1:L PR[91] R[100]mm/sec CNT100;
   1:  PR[GP1:91,1] = PR[GP1:90,1] + -52.077;
   1:  PR[GP1:91,2] = PR[GP1:90,2] + 3.054;
   1:L PR[91] R[100]mm/sec CNT100;
   1:  PR[GP1:91,1] = PR[GP1:90,1] + -52.511;
   1:  PR[GP1:91,2] = PR[GP1:90,2] + -0.059;
   1:L PR[91] R[100]mm/sec CNT100;
   1:  PR[GP1:91,1] = PR[GP1:90,1] + -50.406;
   1:  PR[GP1:91,2] = PR[GP1:90,2] + -11.569;
   1:L PR[91] R[100]mm/sec CNT100;
   1:  PR[GP1:91,1] = PR[GP1:90,1] + -49.944;
   1:  PR[GP1:91,2] = PR[GP1:90,2] + -14.877;
   1:L PR[91] R[100]mm/sec CNT100;
   1:  PR[GP1:91,1] = PR[GP1:90,1] + -48.616;
   1:  PR[GP1:91,2] = PR[GP1:90,2] + -17.886;
   1:L PR[91] R[100]mm/sec CNT100;
   1:  PR[GP1:91,1] = PR[GP1:90,1] + -42.628;
   1:  PR[GP1:91,2] = PR[GP1:90,2] + -27.891;
   1:L PR[91] R[100]mm/sec CNT100;
   1:  PR[GP1:91,1] = PR[GP1:90,1] + -40.336;
   1:  PR[GP1:91,2] = PR[GP1:90,2] + -30.652;
   1:L PR[91] R[100]mm/sec CNT100;
   1:  PR[GP1:91,1] = PR[GP1:90,1] + -31.552;
   1:  PR[GP1:91,2] = PR[GP1:90,2] + -37.697;
   1:L PR[91] R[100]mm/sec CNT100;
   1:  PR[GP1:91,1] = PR[GP1:90,1] + -28.649;
   1:  PR[GP1:91,2] = PR[GP1:90,2] + -39.753;
   1:L PR[91] R[100]mm/sec CNT100;
   1:  PR[GP1:91,1] = PR[GP1:90,1] + -25.327;
   1:  PR[GP1:91,2] = PR[GP1:90,2] + -41.040;
   1:L PR[91] R[100]mm/sec CNT100;
   1:  PR[GP1:91,1] = PR[GP1:90,1] + -14.845;
   1:  PR[GP1:91,2] = PR[GP1:90,2] + -44.569;
   1:L PR[91] R[100]mm/sec CNT100;
   1:  PR[GP1:91,1] = PR[GP1:90,1] + -10.924;
   1:  PR[GP1:91,2] = PR[GP1:90,2] + -45.055;
   1:L PR[91] R[100]mm/sec CNT100;
   1:  PR[GP1:91,1] = PR[GP1:90,1] + -3.925;
   1:  PR[GP1:91,2] = PR[GP1:90,2] + -44.904;
   1:L PR[91] R[100]mm/sec CNT100;
   1:  PR[GP1:91,1] = PR[GP1:90,1] + -0.514;
   1:  PR[GP1:91,2] = PR[GP1:90,2] + -44.816;
   1:L PR[91] R[100]mm/sec CNT100;
   1:  PR[GP1:91,1] = PR[GP1:90,1] + 0.727;
   1:L PR[91] R[100]mm/sec CNT100;
   1:  PR[GP1:91,1] = PR[GP1:90,1] + 4.138;
   1:  PR[GP1:91,2] = PR[GP1:90,2] + -44.904;
   1:L PR[91] R[100]mm/sec CNT100;
   1:  PR[GP1:91,1] = PR[GP1:90,1] + 11.138;
   1:  PR[GP1:91,2] = PR[GP1:90,2] + -45.055;
   1:L PR[91] R[100]mm/sec CNT100;
   1:  PR[GP1:91,1] = PR[GP1:90,1] + 15.059;
   1:  PR[GP1:91,2] = PR[GP1:90,2] + -44.569;
   1:L PR[91] R[100]mm/sec CNT100;
   1:  PR[GP1:91,1] = PR[GP1:90,1] + 25.541;
   1:  PR[GP1:91,2] = PR[GP1:90,2] + -41.040;
   1:L PR[91] R[100]mm/sec CNT100;
   1:  PR[GP1:91,1] = PR[GP1:90,1] + 28.847;
   1:  PR[GP1:91,2] = PR[GP1:90,2] + -39.759;
   1:L PR[91] R[100]mm/sec CNT100;
   1:  PR[GP1:91,1] = PR[GP1:90,1] + 37.928;
   1:  PR[GP1:91,2] = PR[GP1:90,2] + -32.500;
   1:L PR[91] R[100]mm/sec CNT100;
   1:  PR[GP1:91,1] = PR[GP1:90,1] + 40.562;
   1:  PR[GP1:91,2] = PR[GP1:90,2] + -30.635;
   1:L PR[91] R[100]mm/sec CNT100;
   1:  PR[GP1:91,1] = PR[GP1:90,1] + 42.842;
   1:  PR[GP1:91,2] = PR[GP1:90,2] + -27.888;
   1:L PR[91] R[100]mm/sec CNT100;
   1:  PR[GP1:91,1] = PR[GP1:90,1] + 48.829;
   1:  PR[GP1:91,2] = PR[GP1:90,2] + -17.890;
   1:L PR[91] R[100]mm/sec CNT100;
   1:  PR[GP1:91,1] = PR[GP1:90,1] + 50.163;
   1:  PR[GP1:91,2] = PR[GP1:90,2] + -14.869;
   1:L PR[91] R[100]mm/sec CNT100;
   1:  PR[GP1:91,1] = PR[GP1:90,1] + 52.290;
   1:  PR[GP1:91,2] = PR[GP1:90,2] + -3.197;
   1:L PR[91] R[100]mm/sec CNT100;
   1:  PR[GP1:91,1] = PR[GP1:90,1] + 52.724;
   1:  PR[GP1:91,2] = PR[GP1:90,2] + -0.085;
   1:L PR[91] R[100]mm/sec CNT100;
   1:  PR[GP1:91,1] = PR[GP1:90,1] + 50.619;
   1:  PR[GP1:91,2] = PR[GP1:90,2] + 11.430;
   1:L PR[91] R[100]mm/sec CNT100;
   1:  PR[GP1:91,1] = PR[GP1:90,1] + 50.158;
   1:  PR[GP1:91,2] = PR[GP1:90,2] + 14.737;
   1:L PR[91] R[100]mm/sec CNT100;
   1:  PR[GP1:91,1] = PR[GP1:90,1] + 48.829;
   1:  PR[GP1:91,2] = PR[GP1:90,2] + 17.746;
   1:L PR[91] R[100]mm/sec CNT100;
   1:  PR[GP1:91,1] = PR[GP1:90,1] + 42.841;
   1:  PR[GP1:91,2] = PR[GP1:90,2] + 27.745;
   1:L PR[91] R[100]mm/sec CNT100;
   1:  PR[GP1:91,1] = PR[GP1:90,1] + 40.549;
   1:  PR[GP1:91,2] = PR[GP1:90,2] + 30.506;
   1:L PR[91] R[100]mm/sec CNT100;
   1:  PR[GP1:91,1] = PR[GP1:90,1] + 31.765;
   1:  PR[GP1:91,2] = PR[GP1:90,2] + 37.553;
   1:L PR[91] R[100]mm/sec CNT100;
   1:  PR[GP1:91,1] = PR[GP1:90,1] + 28.861;
   1:  PR[GP1:91,2] = PR[GP1:90,2] + 39.610;
   1:L PR[91] R[100]mm/sec CNT100;
   1:  PR[GP1:91,1] = PR[GP1:90,1] + 25.539;
   1:  PR[GP1:91,2] = PR[GP1:90,2] + 40.897;
   1:L PR[91] R[100]mm/sec CNT100;
   1:  PR[GP1:91,1] = PR[GP1:90,1] + 15.056;
   1:  PR[GP1:91,2] = PR[GP1:90,2] + 44.425;
   1:L PR[91] R[100]mm/sec CNT100;
   1:  PR[GP1:91,1] = PR[GP1:90,1] + 11.135;
   1:  PR[GP1:91,2] = PR[GP1:90,2] + 44.911;
   1:L PR[91] R[100]mm/sec CNT100;
   1:  PR[GP1:91,1] = PR[GP1:90,1] + 4.159;
   1:  PR[GP1:91,2] = PR[GP1:90,2] + 44.761;
   1:L PR[91] R[100]mm/sec CNT100;
   1:  PR[GP1:91,1] = PR[GP1:90,1] + 0.727;
   1:  PR[GP1:91,2] = PR[GP1:90,2] + 44.671;
   1:L PR[91] R[100]mm/sec CNT100;
   1:  ! -- Layer/Ebene 181 -- !;
   1:  PR[91] = PR[90];
   1:  PR[GP1:91,1] = PR[GP1:90,1] + -0.490;
   1:  PR[GP1:91,2] = PR[GP1:90,2] + 44.831;
   1:  PR[GP1:91,3] = PR[GP1:90,3] + 110.715;
   1:L PR[91] R[100]mm/sec CNT100;
   1:  PR[GP1:91,1] = PR[GP1:90,1] + -10.551;
   1:  PR[GP1:91,2] = PR[GP1:90,2] + 45.059;
   1:L PR[91] R[100]mm/sec CNT100;
   1:  PR[GP1:91,1] = PR[GP1:90,1] + -14.745;
   1:  PR[GP1:91,2] = PR[GP1:90,2] + 44.539;
   1:L PR[91] R[100]mm/sec CNT100;
   1:  PR[GP1:91,1] = PR[GP1:90,1] + -24.875;
   1:  PR[GP1:91,2] = PR[GP1:90,2] + 41.130;
   1:L PR[91] R[100]mm/sec CNT100;
   1:  PR[GP1:91,1] = PR[GP1:90,1] + -28.450;
   1:  PR[GP1:91,2] = PR[GP1:90,2] + 39.745;
   1:L PR[91] R[100]mm/sec CNT100;
   1:  PR[GP1:91,1] = PR[GP1:90,1] + -37.226;
   1:  PR[GP1:91,2] = PR[GP1:90,2] + 32.733;
   1:L PR[91] R[100]mm/sec CNT100;
   1:  PR[GP1:91,1] = PR[GP1:90,1] + -40.106;
   1:  PR[GP1:91,2] = PR[GP1:90,2] + 30.694;
   1:L PR[91] R[100]mm/sec CNT100;
   1:  PR[GP1:91,1] = PR[GP1:90,1] + -42.603;
   1:  PR[GP1:91,2] = PR[GP1:90,2] + 27.686;
   1:L PR[91] R[100]mm/sec CNT100;
   1:  PR[GP1:91,1] = PR[GP1:90,1] + -48.390;
   1:  PR[GP1:91,2] = PR[GP1:90,2] + 18.019;
   1:L PR[91] R[100]mm/sec CNT100;
   1:  PR[GP1:91,1] = PR[GP1:90,1] + -49.864;
   1:  PR[GP1:91,2] = PR[GP1:90,2] + 14.679;
   1:L PR[91] R[100]mm/sec CNT100;
   1:  PR[GP1:91,1] = PR[GP1:90,1] + -51.920;
   1:  PR[GP1:91,2] = PR[GP1:90,2] + 3.404;
   1:L PR[91] R[100]mm/sec CNT100;
   1:  PR[GP1:91,1] = PR[GP1:90,1] + -52.403;
   1:  PR[GP1:91,2] = PR[GP1:90,2] + -0.059;
   1:L PR[91] R[100]mm/sec CNT100;
   1:  PR[GP1:91,1] = PR[GP1:90,1] + -50.369;
   1:  PR[GP1:91,2] = PR[GP1:90,2] + -11.181;
   1:L PR[91] R[100]mm/sec CNT100;
   1:  PR[GP1:91,1] = PR[GP1:90,1] + -49.859;
   1:  PR[GP1:91,2] = PR[GP1:90,2] + -14.834;
   1:L PR[91] R[100]mm/sec CNT100;
   1:  PR[GP1:91,1] = PR[GP1:90,1] + -48.390;
   1:  PR[GP1:91,2] = PR[GP1:90,2] + -18.162;
   1:L PR[91] R[100]mm/sec CNT100;
   1:  PR[GP1:91,1] = PR[GP1:90,1] + -42.604;
   1:  PR[GP1:91,2] = PR[GP1:90,2] + -27.829;
   1:L PR[91] R[100]mm/sec CNT100;
   1:  PR[GP1:91,1] = PR[GP1:90,1] + -40.095;
   1:  PR[GP1:91,2] = PR[GP1:90,2] + -30.851;
   1:L PR[91] R[100]mm/sec CNT100;
   1:  PR[GP1:91,1] = PR[GP1:90,1] + -31.608;
   1:  PR[GP1:91,2] = PR[GP1:90,2] + -37.658;
   1:L PR[91] R[100]mm/sec CNT100;
   1:  PR[GP1:91,1] = PR[GP1:90,1] + -28.468;
   1:  PR[GP1:91,2] = PR[GP1:90,2] + -39.881;
   1:L PR[91] R[100]mm/sec CNT100;
   1:  PR[GP1:91,1] = PR[GP1:90,1] + -24.877;
   1:  PR[GP1:91,2] = PR[GP1:90,2] + -41.273;
   1:L PR[91] R[100]mm/sec CNT100;
   1:  PR[GP1:91,1] = PR[GP1:90,1] + -14.748;
   1:  PR[GP1:91,2] = PR[GP1:90,2] + -44.683;
   1:L PR[91] R[100]mm/sec CNT100;
   1:  PR[GP1:91,1] = PR[GP1:90,1] + -10.553;
   1:  PR[GP1:91,2] = PR[GP1:90,2] + -45.203;
   1:L PR[91] R[100]mm/sec CNT100;
   1:  PR[GP1:91,1] = PR[GP1:90,1] + -0.490;
   1:  PR[GP1:91,2] = PR[GP1:90,2] + -44.975;
   1:L PR[91] R[100]mm/sec CNT100;
   1:  PR[GP1:91,1] = PR[GP1:90,1] + 0.703;
   1:L PR[91] R[100]mm/sec CNT100;
   1:  PR[GP1:91,1] = PR[GP1:90,1] + 10.767;
   1:  PR[GP1:91,2] = PR[GP1:90,2] + -45.203;
   1:L PR[91] R[100]mm/sec CNT100;
   1:  PR[GP1:91,1] = PR[GP1:90,1] + 14.962;
   1:  PR[GP1:91,2] = PR[GP1:90,2] + -44.683;
   1:L PR[91] R[100]mm/sec CNT100;
   1:  PR[GP1:91,1] = PR[GP1:90,1] + 25.091;
   1:  PR[GP1:91,2] = PR[GP1:90,2] + -41.273;
   1:L PR[91] R[100]mm/sec CNT100;
   1:  PR[GP1:91,1] = PR[GP1:90,1] + 28.666;
   1:  PR[GP1:91,2] = PR[GP1:90,2] + -39.888;
   1:L PR[91] R[100]mm/sec CNT100;
   1:  PR[GP1:91,1] = PR[GP1:90,1] + 37.441;
   1:  PR[GP1:91,2] = PR[GP1:90,2] + -32.873;
   1:L PR[91] R[100]mm/sec CNT100;
   1:  PR[GP1:91,1] = PR[GP1:90,1] + 40.321;
   1:  PR[GP1:91,2] = PR[GP1:90,2] + -30.834;
   1:L PR[91] R[100]mm/sec CNT100;
   1:  PR[GP1:91,1] = PR[GP1:90,1] + 42.818;
   1:  PR[GP1:91,2] = PR[GP1:90,2] + -27.826;
   1:L PR[91] R[100]mm/sec CNT100;
   1:  PR[GP1:91,1] = PR[GP1:90,1] + 48.603;
   1:  PR[GP1:91,2] = PR[GP1:90,2] + -18.165;
   1:L PR[91] R[100]mm/sec CNT100;
   1:  PR[GP1:91,1] = PR[GP1:90,1] + 50.078;
   1:  PR[GP1:91,2] = PR[GP1:90,2] + -14.826;
   1:L PR[91] R[100]mm/sec CNT100;
   1:  PR[GP1:91,1] = PR[GP1:90,1] + 52.133;
   1:  PR[GP1:91,2] = PR[GP1:90,2] + -3.548;
   1:L PR[91] R[100]mm/sec CNT100;
   1:  PR[GP1:91,1] = PR[GP1:90,1] + 52.616;
   1:  PR[GP1:91,2] = PR[GP1:90,2] + -0.085;
   1:L PR[91] R[100]mm/sec CNT100;
   1:  PR[GP1:91,1] = PR[GP1:90,1] + 50.582;
   1:  PR[GP1:91,2] = PR[GP1:90,2] + 11.041;
   1:L PR[91] R[100]mm/sec CNT100;
   1:  PR[GP1:91,1] = PR[GP1:90,1] + 50.072;
   1:  PR[GP1:91,2] = PR[GP1:90,2] + 14.694;
   1:L PR[91] R[100]mm/sec CNT100;
   1:  PR[GP1:91,1] = PR[GP1:90,1] + 48.603;
   1:  PR[GP1:91,2] = PR[GP1:90,2] + 18.022;
   1:L PR[91] R[100]mm/sec CNT100;
   1:  PR[GP1:91,1] = PR[GP1:90,1] + 42.817;
   1:  PR[GP1:91,2] = PR[GP1:90,2] + 27.683;
   1:L PR[91] R[100]mm/sec CNT100;
   1:  PR[GP1:91,1] = PR[GP1:90,1] + 40.309;
   1:  PR[GP1:91,2] = PR[GP1:90,2] + 30.705;
   1:L PR[91] R[100]mm/sec CNT100;
   1:  PR[GP1:91,1] = PR[GP1:90,1] + 31.821;
   1:  PR[GP1:91,2] = PR[GP1:90,2] + 37.514;
   1:L PR[91] R[100]mm/sec CNT100;
   1:  PR[GP1:91,1] = PR[GP1:90,1] + 28.681;
   1:  PR[GP1:91,2] = PR[GP1:90,2] + 39.738;
   1:L PR[91] R[100]mm/sec CNT100;
   1:  PR[GP1:91,1] = PR[GP1:90,1] + 25.089;
   1:  PR[GP1:91,2] = PR[GP1:90,2] + 41.130;
   1:L PR[91] R[100]mm/sec CNT100;
   1:  PR[GP1:91,1] = PR[GP1:90,1] + 14.960;
   1:  PR[GP1:91,2] = PR[GP1:90,2] + 44.539;
   1:L PR[91] R[100]mm/sec CNT100;
   1:  PR[GP1:91,1] = PR[GP1:90,1] + 10.764;
   1:  PR[GP1:91,2] = PR[GP1:90,2] + 45.059;
   1:L PR[91] R[100]mm/sec CNT100;
   1:  PR[GP1:91,1] = PR[GP1:90,1] + 0.703;
   1:  PR[GP1:91,2] = PR[GP1:90,2] + 44.831;
   1:L PR[91] R[100]mm/sec CNT100;
   1:  ! -- Layer/Ebene 182 -- !;
   1:  PR[91] = PR[90];
   1:  PR[GP1:91,1] = PR[GP1:90,1] + -0.467;
   1:  PR[GP1:91,2] = PR[GP1:90,2] + 44.990;
   1:  PR[GP1:91,3] = PR[GP1:90,3] + 111.325;
   1:L PR[91] R[100]mm/sec CNT100;
   1:  PR[GP1:91,1] = PR[GP1:90,1] + -10.180;
   1:  PR[GP1:91,2] = PR[GP1:90,2] + 45.207;
   1:L PR[91] R[100]mm/sec CNT100;
   1:  PR[GP1:91,1] = PR[GP1:90,1] + -14.649;
   1:  PR[GP1:91,2] = PR[GP1:90,2] + 44.653;
   1:L PR[91] R[100]mm/sec CNT100;
   1:  PR[GP1:91,1] = PR[GP1:90,1] + -24.425;
   1:  PR[GP1:91,2] = PR[GP1:90,2] + 41.363;
   1:L PR[91] R[100]mm/sec CNT100;
   1:  PR[GP1:91,1] = PR[GP1:90,1] + -28.270;
   1:  PR[GP1:91,2] = PR[GP1:90,2] + 39.873;
   1:L PR[91] R[100]mm/sec CNT100;
   1:  PR[GP1:91,1] = PR[GP1:90,1] + -36.740;
   1:  PR[GP1:91,2] = PR[GP1:90,2] + 33.106;
   1:L PR[91] R[100]mm/sec CNT100;
   1:  PR[GP1:91,1] = PR[GP1:90,1] + -39.865;
   1:  PR[GP1:91,2] = PR[GP1:90,2] + 30.893;
   1:L PR[91] R[100]mm/sec CNT100;
   1:  PR[GP1:91,1] = PR[GP1:90,1] + -42.579;
   1:  PR[GP1:91,2] = PR[GP1:90,2] + 27.624;
   1:L PR[91] R[100]mm/sec CNT100;
   1:  PR[GP1:91,1] = PR[GP1:90,1] + -48.164;
   1:  PR[GP1:91,2] = PR[GP1:90,2] + 18.294;
   1:L PR[91] R[100]mm/sec CNT100;
   1:  PR[GP1:91,1] = PR[GP1:90,1] + -49.779;
   1:  PR[GP1:91,2] = PR[GP1:90,2] + 14.636;
   1:L PR[91] R[100]mm/sec CNT100;
   1:  PR[GP1:91,1] = PR[GP1:90,1] + -51.763;
   1:  PR[GP1:91,2] = PR[GP1:90,2] + 3.755;
   1:L PR[91] R[100]mm/sec CNT100;
   1:  PR[GP1:91,1] = PR[GP1:90,1] + -52.295;
   1:  PR[GP1:91,2] = PR[GP1:90,2] + -0.059;
   1:L PR[91] R[100]mm/sec CNT100;
   1:  PR[GP1:91,1] = PR[GP1:90,1] + -50.332;
   1:  PR[GP1:91,2] = PR[GP1:90,2] + -10.792;
   1:L PR[91] R[100]mm/sec CNT100;
   1:  PR[GP1:91,1] = PR[GP1:90,1] + -49.774;
   1:  PR[GP1:91,2] = PR[GP1:90,2] + -14.791;
   1:L PR[91] R[100]mm/sec CNT100;
   1:  PR[GP1:91,1] = PR[GP1:90,1] + -48.164;
   1:  PR[GP1:91,2] = PR[GP1:90,2] + -18.438;
   1:L PR[91] R[100]mm/sec CNT100;
   1:  PR[GP1:91,1] = PR[GP1:90,1] + -42.580;
   1:  PR[GP1:91,2] = PR[GP1:90,2] + -27.767;
   1:L PR[91] R[100]mm/sec CNT100;
   1:  PR[GP1:91,1] = PR[GP1:90,1] + -39.855;
   1:  PR[GP1:91,2] = PR[GP1:90,2] + -31.050;
   1:L PR[91] R[100]mm/sec CNT100;
   1:  PR[GP1:91,1] = PR[GP1:90,1] + -31.664;
   1:  PR[GP1:91,2] = PR[GP1:90,2] + -37.619;
   1:L PR[91] R[100]mm/sec CNT100;
   1:  PR[GP1:91,1] = PR[GP1:90,1] + -28.288;
   1:  PR[GP1:91,2] = PR[GP1:90,2] + -40.010;
   1:L PR[91] R[100]mm/sec CNT100;
   1:  PR[GP1:91,1] = PR[GP1:90,1] + -24.426;
   1:  PR[GP1:91,2] = PR[GP1:90,2] + -41.506;
   1:L PR[91] R[100]mm/sec CNT100;
   1:  PR[GP1:91,1] = PR[GP1:90,1] + -14.651;
   1:  PR[GP1:91,2] = PR[GP1:90,2] + -44.797;
   1:L PR[91] R[100]mm/sec CNT100;
   1:  PR[GP1:91,1] = PR[GP1:90,1] + -10.183;
   1:  PR[GP1:91,2] = PR[GP1:90,2] + -45.351;
   1:L PR[91] R[100]mm/sec CNT100;
   1:  PR[GP1:91,1] = PR[GP1:90,1] + -0.468;
   1:  PR[GP1:91,2] = PR[GP1:90,2] + -45.134;
   1:L PR[91] R[100]mm/sec CNT100;
   1:  PR[GP1:91,1] = PR[GP1:90,1] + 0.681;
   1:L PR[91] R[100]mm/sec CNT100;
   1:  PR[GP1:91,1] = PR[GP1:90,1] + 10.396;
   1:  PR[GP1:91,2] = PR[GP1:90,2] + -45.351;
   1:L PR[91] R[100]mm/sec CNT100;
   1:  PR[GP1:91,1] = PR[GP1:90,1] + 14.865;
   1:  PR[GP1:91,2] = PR[GP1:90,2] + -44.797;
   1:L PR[91] R[100]mm/sec CNT100;
   1:  PR[GP1:91,1] = PR[GP1:90,1] + 24.640;
   1:  PR[GP1:91,2] = PR[GP1:90,2] + -41.506;
   1:L PR[91] R[100]mm/sec CNT100;
   1:  PR[GP1:91,1] = PR[GP1:90,1] + 28.486;
   1:  PR[GP1:91,2] = PR[GP1:90,2] + -40.016;
   1:L PR[91] R[100]mm/sec CNT100;
   1:  PR[GP1:91,1] = PR[GP1:90,1] + 36.954;
   1:  PR[GP1:91,2] = PR[GP1:90,2] + -33.247;
   1:L PR[91] R[100]mm/sec CNT100;
   1:  PR[GP1:91,1] = PR[GP1:90,1] + 40.081;
   1:  PR[GP1:91,2] = PR[GP1:90,2] + -31.033;
   1:L PR[91] R[100]mm/sec CNT100;
   1:  PR[GP1:91,1] = PR[GP1:90,1] + 42.794;
   1:  PR[GP1:91,2] = PR[GP1:90,2] + -27.764;
   1:L PR[91] R[100]mm/sec CNT100;
   1:  PR[GP1:91,1] = PR[GP1:90,1] + 48.377;
   1:  PR[GP1:91,2] = PR[GP1:90,2] + -18.441;
   1:L PR[91] R[100]mm/sec CNT100;
   1:  PR[GP1:91,1] = PR[GP1:90,1] + 49.993;
   1:  PR[GP1:91,2] = PR[GP1:90,2] + -14.782;
   1:L PR[91] R[100]mm/sec CNT100;
   1:  PR[GP1:91,1] = PR[GP1:90,1] + 51.976;
   1:  PR[GP1:91,2] = PR[GP1:90,2] + -3.898;
   1:L PR[91] R[100]mm/sec CNT100;
   1:  PR[GP1:91,1] = PR[GP1:90,1] + 52.508;
   1:  PR[GP1:91,2] = PR[GP1:90,2] + -0.085;
   1:L PR[91] R[100]mm/sec CNT100;
   1:  PR[GP1:91,1] = PR[GP1:90,1] + 50.545;
   1:  PR[GP1:91,2] = PR[GP1:90,2] + 10.653;
   1:L PR[91] R[100]mm/sec CNT100;
   1:  PR[GP1:91,1] = PR[GP1:90,1] + 49.987;
   1:  PR[GP1:91,2] = PR[GP1:90,2] + 14.651;
   1:L PR[91] R[100]mm/sec CNT100;
   1:  PR[GP1:91,1] = PR[GP1:90,1] + 48.377;
   1:  PR[GP1:91,2] = PR[GP1:90,2] + 18.297;
   1:L PR[91] R[100]mm/sec CNT100;
   1:  PR[GP1:91,1] = PR[GP1:90,1] + 42.793;
   1:  PR[GP1:91,2] = PR[GP1:90,2] + 27.621;
   1:L PR[91] R[100]mm/sec CNT100;
   1:  PR[GP1:91,1] = PR[GP1:90,1] + 40.068;
   1:  PR[GP1:91,2] = PR[GP1:90,2] + 30.904;
   1:L PR[91] R[100]mm/sec CNT100;
   1:  PR[GP1:91,1] = PR[GP1:90,1] + 31.877;
   1:  PR[GP1:91,2] = PR[GP1:90,2] + 37.476;
   1:L PR[91] R[100]mm/sec CNT100;
   1:  PR[GP1:91,1] = PR[GP1:90,1] + 28.501;
   1:  PR[GP1:91,2] = PR[GP1:90,2] + 39.867;
   1:L PR[91] R[100]mm/sec CNT100;
   1:  PR[GP1:91,1] = PR[GP1:90,1] + 24.638;
   1:  PR[GP1:91,2] = PR[GP1:90,2] + 41.363;
   1:L PR[91] R[100]mm/sec CNT100;
   1:  PR[GP1:91,1] = PR[GP1:90,1] + 14.863;
   1:  PR[GP1:91,2] = PR[GP1:90,2] + 44.654;
   1:L PR[91] R[100]mm/sec CNT100;
   1:  PR[GP1:91,1] = PR[GP1:90,1] + 10.394;
   1:  PR[GP1:91,2] = PR[GP1:90,2] + 45.207;
   1:L PR[91] R[100]mm/sec CNT100;
   1:  PR[GP1:91,1] = PR[GP1:90,1] + 0.680;
   1:  PR[GP1:91,2] = PR[GP1:90,2] + 44.990;
   1:L PR[91] R[100]mm/sec CNT100;
   1:  ! -- Layer/Ebene 183 -- !;
   1:  PR[91] = PR[90];
   1:  PR[GP1:91,1] = PR[GP1:90,1] + -0.445;
   1:  PR[GP1:91,2] = PR[GP1:90,2] + 45.149;
   1:  PR[GP1:91,3] = PR[GP1:90,3] + 111.935;
   1:L PR[91] R[100]mm/sec CNT100;
   1:  PR[GP1:91,1] = PR[GP1:90,1] + -9.809;
   1:  PR[GP1:91,2] = PR[GP1:90,2] + 45.355;
   1:L PR[91] R[100]mm/sec CNT100;
   1:  PR[GP1:91,1] = PR[GP1:90,1] + -14.552;
   1:  PR[GP1:91,2] = PR[GP1:90,2] + 44.768;
   1:L PR[91] R[100]mm/sec CNT100;
   1:  PR[GP1:91,1] = PR[GP1:90,1] + -23.974;
   1:  PR[GP1:91,2] = PR[GP1:90,2] + 41.597;
   1:L PR[91] R[100]mm/sec CNT100;
   1:  PR[GP1:91,1] = PR[GP1:90,1] + -28.089;
   1:  PR[GP1:91,2] = PR[GP1:90,2] + 40.002;
   1:L PR[91] R[100]mm/sec CNT100;
   1:  PR[GP1:91,1] = PR[GP1:90,1] + -36.253;
   1:  PR[GP1:91,2] = PR[GP1:90,2] + 33.479;
   1:L PR[91] R[100]mm/sec CNT100;
   1:  PR[GP1:91,1] = PR[GP1:90,1] + -39.625;
   1:  PR[GP1:91,2] = PR[GP1:90,2] + 31.092;
   1:L PR[91] R[100]mm/sec CNT100;
   1:  PR[GP1:91,1] = PR[GP1:90,1] + -42.555;
   1:  PR[GP1:91,2] = PR[GP1:90,2] + 27.562;
   1:L PR[91] R[100]mm/sec CNT100;
   1:  PR[GP1:91,1] = PR[GP1:90,1] + -47.938;
   1:  PR[GP1:91,2] = PR[GP1:90,2] + 18.570;
   1:L PR[91] R[100]mm/sec CNT100;
   1:  PR[GP1:91,1] = PR[GP1:90,1] + -49.694;
   1:  PR[GP1:91,2] = PR[GP1:90,2] + 14.592;
   1:L PR[91] R[100]mm/sec CNT100;
   1:  PR[GP1:91,1] = PR[GP1:90,1] + -51.606;
   1:  PR[GP1:91,2] = PR[GP1:90,2] + 4.105;
   1:L PR[91] R[100]mm/sec CNT100;
   1:  PR[GP1:91,1] = PR[GP1:90,1] + -52.187;
   1:  PR[GP1:91,2] = PR[GP1:90,2] + -0.059;
   1:L PR[91] R[100]mm/sec CNT100;
   1:  PR[GP1:91,1] = PR[GP1:90,1] + -50.295;
   1:  PR[GP1:91,2] = PR[GP1:90,2] + -10.404;
   1:L PR[91] R[100]mm/sec CNT100;
   1:  PR[GP1:91,1] = PR[GP1:90,1] + -49.689;
   1:  PR[GP1:91,2] = PR[GP1:90,2] + -14.747;
   1:L PR[91] R[100]mm/sec CNT100;
   1:  PR[GP1:91,1] = PR[GP1:90,1] + -47.938;
   1:  PR[GP1:91,2] = PR[GP1:90,2] + -18.713;
   1:L PR[91] R[100]mm/sec CNT100;
   1:  PR[GP1:91,1] = PR[GP1:90,1] + -42.556;
   1:  PR[GP1:91,2] = PR[GP1:90,2] + -27.705;
   1:L PR[91] R[100]mm/sec CNT100;
   1:  PR[GP1:91,1] = PR[GP1:90,1] + -39.614;
   1:  PR[GP1:91,2] = PR[GP1:90,2] + -31.248;
   1:L PR[91] R[100]mm/sec CNT100;
   1:  PR[GP1:91,1] = PR[GP1:90,1] + -31.720;
   1:  PR[GP1:91,2] = PR[GP1:90,2] + -37.580;
   1:L PR[91] R[100]mm/sec CNT100;
   1:  PR[GP1:91,1] = PR[GP1:90,1] + -28.108;
   1:  PR[GP1:91,2] = PR[GP1:90,2] + -40.138;
   1:L PR[91] R[100]mm/sec CNT100;
   1:  PR[GP1:91,1] = PR[GP1:90,1] + -23.976;
   1:  PR[GP1:91,2] = PR[GP1:90,2] + -41.740;
   1:L PR[91] R[100]mm/sec CNT100;
   1:  PR[GP1:91,1] = PR[GP1:90,1] + -14.555;
   1:  PR[GP1:91,2] = PR[GP1:90,2] + -44.911;
   1:L PR[91] R[100]mm/sec CNT100;
   1:  PR[GP1:91,1] = PR[GP1:90,1] + -9.812;
   1:  PR[GP1:91,2] = PR[GP1:90,2] + -45.499;
   1:L PR[91] R[100]mm/sec CNT100;
   1:  PR[GP1:91,1] = PR[GP1:90,1] + -0.445;
   1:  PR[GP1:91,2] = PR[GP1:90,2] + -45.293;
   1:L PR[91] R[100]mm/sec CNT100;
   1:  PR[GP1:91,1] = PR[GP1:90,1] + 0.658;
   1:L PR[91] R[100]mm/sec CNT100;
   1:  PR[GP1:91,1] = PR[GP1:90,1] + 10.025;
   1:  PR[GP1:91,2] = PR[GP1:90,2] + -45.499;
   1:L PR[91] R[100]mm/sec CNT100;
   1:  PR[GP1:91,1] = PR[GP1:90,1] + 14.768;
   1:  PR[GP1:91,2] = PR[GP1:90,2] + -44.911;
   1:L PR[91] R[100]mm/sec CNT100;
   1:  PR[GP1:91,1] = PR[GP1:90,1] + 24.190;
   1:  PR[GP1:91,2] = PR[GP1:90,2] + -41.739;
   1:L PR[91] R[100]mm/sec CNT100;
   1:  PR[GP1:91,1] = PR[GP1:90,1] + 28.305;
   1:  PR[GP1:91,2] = PR[GP1:90,2] + -40.145;
   1:L PR[91] R[100]mm/sec CNT100;
   1:  PR[GP1:91,1] = PR[GP1:90,1] + 36.468;
   1:  PR[GP1:91,2] = PR[GP1:90,2] + -33.620;
   1:L PR[91] R[100]mm/sec CNT100;
   1:  PR[GP1:91,1] = PR[GP1:90,1] + 39.840;
   1:  PR[GP1:91,2] = PR[GP1:90,2] + -31.232;
   1:L PR[91] R[100]mm/sec CNT100;
   1:  PR[GP1:91,1] = PR[GP1:90,1] + 42.770;
   1:  PR[GP1:91,2] = PR[GP1:90,2] + -27.702;
   1:L PR[91] R[100]mm/sec CNT100;
   1:  PR[GP1:91,1] = PR[GP1:90,1] + 48.151;
   1:  PR[GP1:91,2] = PR[GP1:90,2] + -18.716;
   1:L PR[91] R[100]mm/sec CNT100;
   1:  PR[GP1:91,1] = PR[GP1:90,1] + 49.907;
   1:  PR[GP1:91,2] = PR[GP1:90,2] + -14.739;
   1:L PR[91] R[100]mm/sec CNT100;
   1:  PR[GP1:91,1] = PR[GP1:90,1] + 51.819;
   1:  PR[GP1:91,2] = PR[GP1:90,2] + -4.249;
   1:L PR[91] R[100]mm/sec CNT100;
   1:  PR[GP1:91,1] = PR[GP1:90,1] + 52.400;
   1:  PR[GP1:91,2] = PR[GP1:90,2] + -0.085;
   1:L PR[91] R[100]mm/sec CNT100;
   1:  PR[GP1:91,1] = PR[GP1:90,1] + 50.508;
   1:  PR[GP1:91,2] = PR[GP1:90,2] + 10.264;
   1:L PR[91] R[100]mm/sec CNT100;
   1:  PR[GP1:91,1] = PR[GP1:90,1] + 49.902;
   1:  PR[GP1:91,2] = PR[GP1:90,2] + 14.607;
   1:L PR[91] R[100]mm/sec CNT100;
   1:  PR[GP1:91,1] = PR[GP1:90,1] + 48.151;
   1:  PR[GP1:91,2] = PR[GP1:90,2] + 18.573;
   1:L PR[91] R[100]mm/sec CNT100;
   1:  PR[GP1:91,1] = PR[GP1:90,1] + 42.769;
   1:  PR[GP1:91,2] = PR[GP1:90,2] + 27.559;
   1:L PR[91] R[100]mm/sec CNT100;
   1:  PR[GP1:91,1] = PR[GP1:90,1] + 39.828;
   1:  PR[GP1:91,2] = PR[GP1:90,2] + 31.103;
   1:L PR[91] R[100]mm/sec CNT100;
   1:  PR[GP1:91,1] = PR[GP1:90,1] + 31.933;
   1:  PR[GP1:91,2] = PR[GP1:90,2] + 37.437;
   1:L PR[91] R[100]mm/sec CNT100;
   1:  PR[GP1:91,1] = PR[GP1:90,1] + 28.320;
   1:  PR[GP1:91,2] = PR[GP1:90,2] + 39.995;
   1:L PR[91] R[100]mm/sec CNT100;
   1:  PR[GP1:91,1] = PR[GP1:90,1] + 24.188;
   1:  PR[GP1:91,2] = PR[GP1:90,2] + 41.596;
   1:L PR[91] R[100]mm/sec CNT100;
   1:  PR[GP1:91,1] = PR[GP1:90,1] + 14.766;
   1:  PR[GP1:91,2] = PR[GP1:90,2] + 44.768;
   1:L PR[91] R[100]mm/sec CNT100;
   1:  PR[GP1:91,1] = PR[GP1:90,1] + 10.023;
   1:  PR[GP1:91,2] = PR[GP1:90,2] + 45.355;
   1:L PR[91] R[100]mm/sec CNT100;
   1:  PR[GP1:91,1] = PR[GP1:90,1] + 0.657;
   1:  PR[GP1:91,2] = PR[GP1:90,2] + 45.149;
   1:L PR[91] R[100]mm/sec CNT100;
   1:  ! -- Layer/Ebene 184 -- !;
   1:  PR[91] = PR[90];
   1:  PR[GP1:91,1] = PR[GP1:90,1] + -0.408;
   1:  PR[GP1:91,2] = PR[GP1:90,2] + 45.309;
   1:  PR[GP1:91,3] = PR[GP1:90,3] + 112.545;
   1:L PR[91] R[100]mm/sec CNT100;
   1:  PR[GP1:91,1] = PR[GP1:90,1] + -9.439;
   1:  PR[GP1:91,2] = PR[GP1:90,2] + 45.503;
   1:L PR[91] R[100]mm/sec CNT100;
   1:  PR[GP1:91,1] = PR[GP1:90,1] + -14.456;
   1:  PR[GP1:91,2] = PR[GP1:90,2] + 44.882;
   1:L PR[91] R[100]mm/sec CNT100;
   1:  PR[GP1:91,1] = PR[GP1:90,1] + -23.524;
   1:  PR[GP1:91,2] = PR[GP1:90,2] + 41.830;
   1:L PR[91] R[100]mm/sec CNT100;
   1:  PR[GP1:91,1] = PR[GP1:90,1] + -27.909;
   1:  PR[GP1:91,2] = PR[GP1:90,2] + 40.130;
   1:L PR[91] R[100]mm/sec CNT100;
   1:  PR[GP1:91,1] = PR[GP1:90,1] + -35.766;
   1:  PR[GP1:91,2] = PR[GP1:90,2] + 33.852;
   1:L PR[91] R[100]mm/sec CNT100;
   1:  PR[GP1:91,1] = PR[GP1:90,1] + -39.384;
   1:  PR[GP1:91,2] = PR[GP1:90,2] + 31.290;
   1:L PR[91] R[100]mm/sec CNT100;
   1:  PR[GP1:91,1] = PR[GP1:90,1] + -42.531;
   1:  PR[GP1:91,2] = PR[GP1:90,2] + 27.500;
   1:L PR[91] R[100]mm/sec CNT100;
   1:  PR[GP1:91,1] = PR[GP1:90,1] + -47.712;
   1:  PR[GP1:91,2] = PR[GP1:90,2] + 18.846;
   1:L PR[91] R[100]mm/sec CNT100;
   1:  PR[GP1:91,1] = PR[GP1:90,1] + -49.608;
   1:  PR[GP1:91,2] = PR[GP1:90,2] + 14.549;
   1:L PR[91] R[100]mm/sec CNT100;
   1:  PR[GP1:91,1] = PR[GP1:90,1] + -51.449;
   1:  PR[GP1:91,2] = PR[GP1:90,2] + 4.456;
   1:L PR[91] R[100]mm/sec CNT100;
   1:  PR[GP1:91,1] = PR[GP1:90,1] + -52.079;
   1:  PR[GP1:91,2] = PR[GP1:90,2] + -0.059;
   1:L PR[91] R[100]mm/sec CNT100;
   1:  PR[GP1:91,1] = PR[GP1:90,1] + -50.258;
   1:  PR[GP1:91,2] = PR[GP1:90,2] + -10.015;
   1:L PR[91] R[100]mm/sec CNT100;
   1:  PR[GP1:91,1] = PR[GP1:90,1] + -49.604;
   1:  PR[GP1:91,2] = PR[GP1:90,2] + -14.704;
   1:L PR[91] R[100]mm/sec CNT100;
   1:  PR[GP1:91,1] = PR[GP1:90,1] + -47.712;
   1:  PR[GP1:91,2] = PR[GP1:90,2] + -18.989;
   1:L PR[91] R[100]mm/sec CNT100;
   1:  PR[GP1:91,1] = PR[GP1:90,1] + -42.532;
   1:  PR[GP1:91,2] = PR[GP1:90,2] + -27.643;
   1:L PR[91] R[100]mm/sec CNT100;
   1:  PR[GP1:91,1] = PR[GP1:90,1] + -39.374;
   1:  PR[GP1:91,2] = PR[GP1:90,2] + -31.447;
   1:L PR[91] R[100]mm/sec CNT100;
   1:  PR[GP1:91,1] = PR[GP1:90,1] + -31.776;
   1:  PR[GP1:91,2] = PR[GP1:90,2] + -37.541;
   1:L PR[91] R[100]mm/sec CNT100;
   1:  PR[GP1:91,1] = PR[GP1:90,1] + -27.927;
   1:  PR[GP1:91,2] = PR[GP1:90,2] + -40.267;
   1:L PR[91] R[100]mm/sec CNT100;
   1:  PR[GP1:91,1] = PR[GP1:90,1] + -23.526;
   1:  PR[GP1:91,2] = PR[GP1:90,2] + -41.973;
   1:L PR[91] R[100]mm/sec CNT100;
   1:  PR[GP1:91,1] = PR[GP1:90,1] + -14.458;
   1:  PR[GP1:91,2] = PR[GP1:90,2] + -45.025;
   1:L PR[91] R[100]mm/sec CNT100;
   1:  PR[GP1:91,1] = PR[GP1:90,1] + -9.441;
   1:  PR[GP1:91,2] = PR[GP1:90,2] + -45.647;
   1:L PR[91] R[100]mm/sec CNT100;
   1:  PR[GP1:91,1] = PR[GP1:90,1] + -0.422;
   1:  PR[GP1:91,2] = PR[GP1:90,2] + -45.453;
   1:L PR[91] R[100]mm/sec CNT100;
   1:  PR[GP1:91,1] = PR[GP1:90,1] + 0.624;
   1:L PR[91] R[100]mm/sec CNT100;
   1:  PR[GP1:91,1] = PR[GP1:90,1] + 9.654;
   1:  PR[GP1:91,2] = PR[GP1:90,2] + -45.647;
   1:L PR[91] R[100]mm/sec CNT100;
   1:  PR[GP1:91,1] = PR[GP1:90,1] + 14.672;
   1:  PR[GP1:91,2] = PR[GP1:90,2] + -45.025;
   1:L PR[91] R[100]mm/sec CNT100;
   1:  PR[GP1:91,1] = PR[GP1:90,1] + 23.739;
   1:  PR[GP1:91,2] = PR[GP1:90,2] + -41.973;
   1:L PR[91] R[100]mm/sec CNT100;
   1:  PR[GP1:91,1] = PR[GP1:90,1] + 28.125;
   1:  PR[GP1:91,2] = PR[GP1:90,2] + -40.273;
   1:L PR[91] R[100]mm/sec CNT100;
   1:  PR[GP1:91,1] = PR[GP1:90,1] + 35.981;
   1:  PR[GP1:91,2] = PR[GP1:90,2] + -33.993;
   1:L PR[91] R[100]mm/sec CNT100;
   1:  PR[GP1:91,1] = PR[GP1:90,1] + 39.600;
   1:  PR[GP1:91,2] = PR[GP1:90,2] + -31.431;
   1:L PR[91] R[100]mm/sec CNT100;
   1:  PR[GP1:91,1] = PR[GP1:90,1] + 42.746;
   1:  PR[GP1:91,2] = PR[GP1:90,2] + -27.641;
   1:L PR[91] R[100]mm/sec CNT100;
   1:  PR[GP1:91,1] = PR[GP1:90,1] + 47.925;
   1:  PR[GP1:91,2] = PR[GP1:90,2] + -18.992;
   1:L PR[91] R[100]mm/sec CNT100;
   1:  PR[GP1:91,1] = PR[GP1:90,1] + 49.822;
   1:  PR[GP1:91,2] = PR[GP1:90,2] + -14.696;
   1:L PR[91] R[100]mm/sec CNT100;
   1:  PR[GP1:91,1] = PR[GP1:90,1] + 51.662;
   1:  PR[GP1:91,2] = PR[GP1:90,2] + -4.600;
   1:L PR[91] R[100]mm/sec CNT100;
   1:  PR[GP1:91,1] = PR[GP1:90,1] + 52.292;
   1:  PR[GP1:91,2] = PR[GP1:90,2] + -0.085;
   1:L PR[91] R[100]mm/sec CNT100;
   1:  PR[GP1:91,1] = PR[GP1:90,1] + 50.471;
   1:  PR[GP1:91,2] = PR[GP1:90,2] + 9.875;
   1:L PR[91] R[100]mm/sec CNT100;
   1:  PR[GP1:91,1] = PR[GP1:90,1] + 49.817;
   1:  PR[GP1:91,2] = PR[GP1:90,2] + 14.564;
   1:L PR[91] R[100]mm/sec CNT100;
   1:  PR[GP1:91,1] = PR[GP1:90,1] + 47.925;
   1:  PR[GP1:91,2] = PR[GP1:90,2] + 18.849;
   1:L PR[91] R[100]mm/sec CNT100;
   1:  PR[GP1:91,1] = PR[GP1:90,1] + 42.746;
   1:  PR[GP1:91,2] = PR[GP1:90,2] + 27.498;
   1:L PR[91] R[100]mm/sec CNT100;
   1:  PR[GP1:91,1] = PR[GP1:90,1] + 39.587;
   1:  PR[GP1:91,2] = PR[GP1:90,2] + 31.302;
   1:L PR[91] R[100]mm/sec CNT100;
   1:  PR[GP1:91,1] = PR[GP1:90,1] + 31.989;
   1:  PR[GP1:91,2] = PR[GP1:90,2] + 37.398;
   1:L PR[91] R[100]mm/sec CNT100;
   1:  PR[GP1:91,1] = PR[GP1:90,1] + 28.140;
   1:  PR[GP1:91,2] = PR[GP1:90,2] + 40.124;
   1:L PR[91] R[100]mm/sec CNT100;
   1:  PR[GP1:91,1] = PR[GP1:90,1] + 23.738;
   1:  PR[GP1:91,2] = PR[GP1:90,2] + 41.830;
   1:L PR[91] R[100]mm/sec CNT100;
   1:  PR[GP1:91,1] = PR[GP1:90,1] + 14.669;
   1:  PR[GP1:91,2] = PR[GP1:90,2] + 44.882;
   1:L PR[91] R[100]mm/sec CNT100;
   1:  PR[GP1:91,1] = PR[GP1:90,1] + 9.652;
   1:  PR[GP1:91,2] = PR[GP1:90,2] + 45.503;
   1:L PR[91] R[100]mm/sec CNT100;
   1:  PR[GP1:91,1] = PR[GP1:90,1] + 0.635;
   1:  PR[GP1:91,2] = PR[GP1:90,2] + 45.309;
   1:L PR[91] R[100]mm/sec CNT100;
   1:  ! -- Layer/Ebene 185 -- !;
   1:  PR[91] = PR[90];
   1:  PR[GP1:91,1] = PR[GP1:90,1] + -0.401;
   1:  PR[GP1:91,2] = PR[GP1:90,2] + 45.465;
   1:  PR[GP1:91,3] = PR[GP1:90,3] + 113.155;
   1:L PR[91] R[100]mm/sec CNT100;
   1:  PR[GP1:91,1] = PR[GP1:90,1] + -9.068;
   1:  PR[GP1:91,2] = PR[GP1:90,2] + 45.651;
   1:L PR[91] R[100]mm/sec CNT100;
   1:  PR[GP1:91,1] = PR[GP1:90,1] + -14.359;
   1:  PR[GP1:91,2] = PR[GP1:90,2] + 44.996;
   1:L PR[91] R[100]mm/sec CNT100;
   1:  PR[GP1:91,1] = PR[GP1:90,1] + -23.074;
   1:  PR[GP1:91,2] = PR[GP1:90,2] + 42.063;
   1:L PR[91] R[100]mm/sec CNT100;
   1:  PR[GP1:91,1] = PR[GP1:90,1] + -27.729;
   1:  PR[GP1:91,2] = PR[GP1:90,2] + 40.259;
   1:L PR[91] R[100]mm/sec CNT100;
   1:  PR[GP1:91,1] = PR[GP1:90,1] + -35.280;
   1:  PR[GP1:91,2] = PR[GP1:90,2] + 34.226;
   1:L PR[91] R[100]mm/sec CNT100;
   1:  PR[GP1:91,1] = PR[GP1:90,1] + -39.144;
   1:  PR[GP1:91,2] = PR[GP1:90,2] + 31.489;
   1:L PR[91] R[100]mm/sec CNT100;
   1:  PR[GP1:91,1] = PR[GP1:90,1] + -42.508;
   1:  PR[GP1:91,2] = PR[GP1:90,2] + 27.438;
   1:L PR[91] R[100]mm/sec CNT100;
   1:  PR[GP1:91,1] = PR[GP1:90,1] + -47.486;
   1:  PR[GP1:91,2] = PR[GP1:90,2] + 19.122;
   1:L PR[91] R[100]mm/sec CNT100;
   1:  PR[GP1:91,1] = PR[GP1:90,1] + -49.523;
   1:  PR[GP1:91,2] = PR[GP1:90,2] + 14.506;
   1:L PR[91] R[100]mm/sec CNT100;
   1:  PR[GP1:91,1] = PR[GP1:90,1] + -51.292;
   1:  PR[GP1:91,2] = PR[GP1:90,2] + 4.807;
   1:L PR[91] R[100]mm/sec CNT100;
   1:  PR[GP1:91,1] = PR[GP1:90,1] + -51.970;
   1:  PR[GP1:91,2] = PR[GP1:90,2] + -0.059;
   1:L PR[91] R[100]mm/sec CNT100;
   1:  PR[GP1:91,1] = PR[GP1:90,1] + -50.221;
   1:  PR[GP1:91,2] = PR[GP1:90,2] + -9.627;
   1:L PR[91] R[100]mm/sec CNT100;
   1:  PR[GP1:91,1] = PR[GP1:90,1] + -49.518;
   1:  PR[GP1:91,2] = PR[GP1:90,2] + -14.661;
   1:L PR[91] R[100]mm/sec CNT100;
   1:  PR[GP1:91,1] = PR[GP1:90,1] + -47.486;
   1:  PR[GP1:91,2] = PR[GP1:90,2] + -19.265;
   1:L PR[91] R[100]mm/sec CNT100;
   1:  PR[GP1:91,1] = PR[GP1:90,1] + -42.508;
   1:  PR[GP1:91,2] = PR[GP1:90,2] + -27.581;
   1:L PR[91] R[100]mm/sec CNT100;
   1:  PR[GP1:91,1] = PR[GP1:90,1] + -39.133;
   1:  PR[GP1:91,2] = PR[GP1:90,2] + -31.646;
   1:L PR[91] R[100]mm/sec CNT100;
   1:  PR[GP1:91,1] = PR[GP1:90,1] + -31.832;
   1:  PR[GP1:91,2] = PR[GP1:90,2] + -37.503;
   1:L PR[91] R[100]mm/sec CNT100;
   1:  PR[GP1:91,1] = PR[GP1:90,1] + -27.747;
   1:  PR[GP1:91,2] = PR[GP1:90,2] + -40.395;
   1:L PR[91] R[100]mm/sec CNT100;
   1:  PR[GP1:91,1] = PR[GP1:90,1] + -23.075;
   1:  PR[GP1:91,2] = PR[GP1:90,2] + -42.206;
   1:L PR[91] R[100]mm/sec CNT100;
   1:  PR[GP1:91,1] = PR[GP1:90,1] + -14.361;
   1:  PR[GP1:91,2] = PR[GP1:90,2] + -45.139;
   1:L PR[91] R[100]mm/sec CNT100;
   1:  PR[GP1:91,1] = PR[GP1:90,1] + -9.070;
   1:  PR[GP1:91,2] = PR[GP1:90,2] + -45.795;
   1:L PR[91] R[100]mm/sec CNT100;
   1:  PR[GP1:91,1] = PR[GP1:90,1] + -0.402;
   1:  PR[GP1:91,2] = PR[GP1:90,2] + -45.609;
   1:L PR[91] R[100]mm/sec CNT100;
   1:  PR[GP1:91,1] = PR[GP1:90,1] + 0.614;
   1:L PR[91] R[100]mm/sec CNT100;
   1:  PR[GP1:91,1] = PR[GP1:90,1] + 9.283;
   1:  PR[GP1:91,2] = PR[GP1:90,2] + -45.795;
   1:L PR[91] R[100]mm/sec CNT100;
   1:  PR[GP1:91,1] = PR[GP1:90,1] + 14.575;
   1:  PR[GP1:91,2] = PR[GP1:90,2] + -45.139;
   1:L PR[91] R[100]mm/sec CNT100;
   1:  PR[GP1:91,1] = PR[GP1:90,1] + 23.289;
   1:  PR[GP1:91,2] = PR[GP1:90,2] + -42.206;
   1:L PR[91] R[100]mm/sec CNT100;
   1:  PR[GP1:91,1] = PR[GP1:90,1] + 27.945;
   1:  PR[GP1:91,2] = PR[GP1:90,2] + -40.402;
   1:L PR[91] R[100]mm/sec CNT100;
   1:  PR[GP1:91,1] = PR[GP1:90,1] + 35.494;
   1:  PR[GP1:91,2] = PR[GP1:90,2] + -34.367;
   1:L PR[91] R[100]mm/sec CNT100;
   1:  PR[GP1:91,1] = PR[GP1:90,1] + 39.359;
   1:  PR[GP1:91,2] = PR[GP1:90,2] + -31.630;
   1:L PR[91] R[100]mm/sec CNT100;
   1:  PR[GP1:91,1] = PR[GP1:90,1] + 42.722;
   1:  PR[GP1:91,2] = PR[GP1:90,2] + -27.579;
   1:L PR[91] R[100]mm/sec CNT100;
   1:  PR[GP1:91,1] = PR[GP1:90,1] + 47.699;
   1:  PR[GP1:91,2] = PR[GP1:90,2] + -19.268;
   1:L PR[91] R[100]mm/sec CNT100;
   1:  PR[GP1:91,1] = PR[GP1:90,1] + 49.737;
   1:  PR[GP1:91,2] = PR[GP1:90,2] + -14.652;
   1:L PR[91] R[100]mm/sec CNT100;
   1:  PR[GP1:91,1] = PR[GP1:90,1] + 51.505;
   1:  PR[GP1:91,2] = PR[GP1:90,2] + -4.950;
   1:L PR[91] R[100]mm/sec CNT100;
   1:  PR[GP1:91,1] = PR[GP1:90,1] + 52.184;
   1:  PR[GP1:91,2] = PR[GP1:90,2] + -0.085;
   1:L PR[91] R[100]mm/sec CNT100;
   1:  PR[GP1:91,1] = PR[GP1:90,1] + 50.434;
   1:  PR[GP1:91,2] = PR[GP1:90,2] + 9.486;
   1:L PR[91] R[100]mm/sec CNT100;
   1:  PR[GP1:91,1] = PR[GP1:90,1] + 49.732;
   1:  PR[GP1:91,2] = PR[GP1:90,2] + 14.520;
   1:L PR[91] R[100]mm/sec CNT100;
   1:  PR[GP1:91,1] = PR[GP1:90,1] + 47.699;
   1:  PR[GP1:91,2] = PR[GP1:90,2] + 19.124;
   1:L PR[91] R[100]mm/sec CNT100;
   1:  PR[GP1:91,1] = PR[GP1:90,1] + 42.722;
   1:  PR[GP1:91,2] = PR[GP1:90,2] + 27.436;
   1:L PR[91] R[100]mm/sec CNT100;
   1:  PR[GP1:91,1] = PR[GP1:90,1] + 39.347;
   1:  PR[GP1:91,2] = PR[GP1:90,2] + 31.501;
   1:L PR[91] R[100]mm/sec CNT100;
   1:  PR[GP1:91,1] = PR[GP1:90,1] + 32.045;
   1:  PR[GP1:91,2] = PR[GP1:90,2] + 37.359;
   1:L PR[91] R[100]mm/sec CNT100;
   1:  PR[GP1:91,1] = PR[GP1:90,1] + 27.960;
   1:  PR[GP1:91,2] = PR[GP1:90,2] + 40.252;
   1:L PR[91] R[100]mm/sec CNT100;
   1:  PR[GP1:91,1] = PR[GP1:90,1] + 23.287;
   1:  PR[GP1:91,2] = PR[GP1:90,2] + 42.063;
   1:L PR[91] R[100]mm/sec CNT100;
   1:  PR[GP1:91,1] = PR[GP1:90,1] + 14.573;
   1:  PR[GP1:91,2] = PR[GP1:90,2] + 44.996;
   1:L PR[91] R[100]mm/sec CNT100;
   1:  PR[GP1:91,1] = PR[GP1:90,1] + 9.281;
   1:  PR[GP1:91,2] = PR[GP1:90,2] + 45.651;
   1:L PR[91] R[100]mm/sec CNT100;
   1:  PR[GP1:91,1] = PR[GP1:90,1] + 0.614;
   1:  PR[GP1:91,2] = PR[GP1:90,2] + 45.465;
   1:L PR[91] R[100]mm/sec CNT100;
   1:  ! -- Layer/Ebene 186 -- !;
   1:  PR[91] = PR[90];
   1:  PR[GP1:91,1] = PR[GP1:90,1] + -0.381;
   1:  PR[GP1:91,2] = PR[GP1:90,2] + 45.620;
   1:  PR[GP1:91,3] = PR[GP1:90,3] + 113.765;
   1:L PR[91] R[100]mm/sec CNT100;
   1:  PR[GP1:91,1] = PR[GP1:90,1] + -8.697;
   1:  PR[GP1:91,2] = PR[GP1:90,2] + 45.799;
   1:L PR[91] R[100]mm/sec CNT100;
   1:  PR[GP1:91,1] = PR[GP1:90,1] + -14.262;
   1:  PR[GP1:91,2] = PR[GP1:90,2] + 45.110;
   1:L PR[91] R[100]mm/sec CNT100;
   1:  PR[GP1:91,1] = PR[GP1:90,1] + -22.623;
   1:  PR[GP1:91,2] = PR[GP1:90,2] + 42.296;
   1:L PR[91] R[100]mm/sec CNT100;
   1:  PR[GP1:91,1] = PR[GP1:90,1] + -27.548;
   1:  PR[GP1:91,2] = PR[GP1:90,2] + 40.387;
   1:L PR[91] R[100]mm/sec CNT100;
   1:  PR[GP1:91,1] = PR[GP1:90,1] + -34.793;
   1:  PR[GP1:91,2] = PR[GP1:90,2] + 34.599;
   1:L PR[91] R[100]mm/sec CNT100;
   1:  PR[GP1:91,1] = PR[GP1:90,1] + -38.903;
   1:  PR[GP1:91,2] = PR[GP1:90,2] + 31.688;
   1:L PR[91] R[100]mm/sec CNT100;
   1:  PR[GP1:91,1] = PR[GP1:90,1] + -42.484;
   1:  PR[GP1:91,2] = PR[GP1:90,2] + 27.376;
   1:L PR[91] R[100]mm/sec CNT100;
   1:  PR[GP1:91,1] = PR[GP1:90,1] + -47.260;
   1:  PR[GP1:91,2] = PR[GP1:90,2] + 19.397;
   1:L PR[91] R[100]mm/sec CNT100;
   1:  PR[GP1:91,1] = PR[GP1:90,1] + -49.438;
   1:  PR[GP1:91,2] = PR[GP1:90,2] + 14.463;
   1:L PR[91] R[100]mm/sec CNT100;
   1:  PR[GP1:91,1] = PR[GP1:90,1] + -51.135;
   1:  PR[GP1:91,2] = PR[GP1:90,2] + 5.157;
   1:L PR[91] R[100]mm/sec CNT100;
   1:  PR[GP1:91,1] = PR[GP1:90,1] + -51.862;
   1:  PR[GP1:91,2] = PR[GP1:90,2] + -0.059;
   1:L PR[91] R[100]mm/sec CNT100;
   1:  PR[GP1:91,1] = PR[GP1:90,1] + -50.184;
   1:  PR[GP1:91,2] = PR[GP1:90,2] + -9.238;
   1:L PR[91] R[100]mm/sec CNT100;
   1:  PR[GP1:91,1] = PR[GP1:90,1] + -49.433;
   1:  PR[GP1:91,2] = PR[GP1:90,2] + -14.618;
   1:L PR[91] R[100]mm/sec CNT100;
   1:  PR[GP1:91,1] = PR[GP1:90,1] + -47.260;
   1:  PR[GP1:91,2] = PR[GP1:90,2] + -19.541;
   1:L PR[91] R[100]mm/sec CNT100;
   1:  PR[GP1:91,1] = PR[GP1:90,1] + -42.485;
   1:  PR[GP1:91,2] = PR[GP1:90,2] + -27.519;
   1:L PR[91] R[100]mm/sec CNT100;
   1:  PR[GP1:91,1] = PR[GP1:90,1] + -38.893;
   1:  PR[GP1:91,2] = PR[GP1:90,2] + -31.845;
   1:L PR[91] R[100]mm/sec CNT100;
   1:  PR[GP1:91,1] = PR[GP1:90,1] + -31.888;
   1:  PR[GP1:91,2] = PR[GP1:90,2] + -37.464;
   1:L PR[91] R[100]mm/sec CNT100;
   1:  PR[GP1:91,1] = PR[GP1:90,1] + -27.567;
   1:  PR[GP1:91,2] = PR[GP1:90,2] + -40.524;
   1:L PR[91] R[100]mm/sec CNT100;
   1:  PR[GP1:91,1] = PR[GP1:90,1] + -22.625;
   1:  PR[GP1:91,2] = PR[GP1:90,2] + -42.439;
   1:L PR[91] R[100]mm/sec CNT100;
   1:  PR[GP1:91,1] = PR[GP1:90,1] + -14.265;
   1:  PR[GP1:91,2] = PR[GP1:90,2] + -45.253;
   1:L PR[91] R[100]mm/sec CNT100;
   1:  PR[GP1:91,1] = PR[GP1:90,1] + -8.700;
   1:  PR[GP1:91,2] = PR[GP1:90,2] + -45.943;
   1:L PR[91] R[100]mm/sec CNT100;
   1:  PR[GP1:91,1] = PR[GP1:90,1] + -0.382;
   1:  PR[GP1:91,2] = PR[GP1:90,2] + -45.764;
   1:L PR[91] R[100]mm/sec CNT100;
   1:  PR[GP1:91,1] = PR[GP1:90,1] + 0.594;
   1:L PR[91] R[100]mm/sec CNT100;
   1:  PR[GP1:91,1] = PR[GP1:90,1] + 8.913;
   1:  PR[GP1:91,2] = PR[GP1:90,2] + -45.943;
   1:L PR[91] R[100]mm/sec CNT100;
   1:  PR[GP1:91,1] = PR[GP1:90,1] + 14.478;
   1:  PR[GP1:91,2] = PR[GP1:90,2] + -45.254;
   1:L PR[91] R[100]mm/sec CNT100;
   1:  PR[GP1:91,1] = PR[GP1:90,1] + 22.838;
   1:  PR[GP1:91,2] = PR[GP1:90,2] + -42.439;
   1:L PR[91] R[100]mm/sec CNT100;
   1:  PR[GP1:91,1] = PR[GP1:90,1] + 27.764;
   1:  PR[GP1:91,2] = PR[GP1:90,2] + -40.530;
   1:L PR[91] R[100]mm/sec CNT100;
   1:  PR[GP1:91,1] = PR[GP1:90,1] + 35.008;
   1:  PR[GP1:91,2] = PR[GP1:90,2] + -34.740;
   1:L PR[91] R[100]mm/sec CNT100;
   1:  PR[GP1:91,1] = PR[GP1:90,1] + 39.119;
   1:  PR[GP1:91,2] = PR[GP1:90,2] + -31.829;
   1:L PR[91] R[100]mm/sec CNT100;
   1:  PR[GP1:91,1] = PR[GP1:90,1] + 42.699;
   1:  PR[GP1:91,2] = PR[GP1:90,2] + -27.517;
   1:L PR[91] R[100]mm/sec CNT100;
   1:  PR[GP1:91,1] = PR[GP1:90,1] + 47.473;
   1:  PR[GP1:91,2] = PR[GP1:90,2] + -19.543;
   1:L PR[91] R[100]mm/sec CNT100;
   1:  PR[GP1:91,1] = PR[GP1:90,1] + 49.652;
   1:  PR[GP1:91,2] = PR[GP1:90,2] + -14.609;
   1:L PR[91] R[100]mm/sec CNT100;
   1:  PR[GP1:91,1] = PR[GP1:90,1] + 51.348;
   1:  PR[GP1:91,2] = PR[GP1:90,2] + -5.301;
   1:L PR[91] R[100]mm/sec CNT100;
   1:  PR[GP1:91,1] = PR[GP1:90,1] + 52.076;
   1:  PR[GP1:91,2] = PR[GP1:90,2] + -0.085;
   1:L PR[91] R[100]mm/sec CNT100;
   1:  PR[GP1:91,1] = PR[GP1:90,1] + 50.397;
   1:  PR[GP1:91,2] = PR[GP1:90,2] + 9.098;
   1:L PR[91] R[100]mm/sec CNT100;
   1:  PR[GP1:91,1] = PR[GP1:90,1] + 49.646;
   1:  PR[GP1:91,2] = PR[GP1:90,2] + 14.477;
   1:L PR[91] R[100]mm/sec CNT100;
   1:  PR[GP1:91,1] = PR[GP1:90,1] + 47.473;
   1:  PR[GP1:91,2] = PR[GP1:90,2] + 19.400;
   1:L PR[91] R[100]mm/sec CNT100;
   1:  PR[GP1:91,1] = PR[GP1:90,1] + 42.698;
   1:  PR[GP1:91,2] = PR[GP1:90,2] + 27.374;
   1:L PR[91] R[100]mm/sec CNT100;
   1:  PR[GP1:91,1] = PR[GP1:90,1] + 39.106;
   1:  PR[GP1:91,2] = PR[GP1:90,2] + 31.700;
   1:L PR[91] R[100]mm/sec CNT100;
   1:  PR[GP1:91,1] = PR[GP1:90,1] + 32.101;
   1:  PR[GP1:91,2] = PR[GP1:90,2] + 37.320;
   1:L PR[91] R[100]mm/sec CNT100;
   1:  PR[GP1:91,1] = PR[GP1:90,1] + 27.779;
   1:  PR[GP1:91,2] = PR[GP1:90,2] + 40.381;
   1:L PR[91] R[100]mm/sec CNT100;
   1:  PR[GP1:91,1] = PR[GP1:90,1] + 22.837;
   1:  PR[GP1:91,2] = PR[GP1:90,2] + 42.296;
   1:L PR[91] R[100]mm/sec CNT100;
   1:  PR[GP1:91,1] = PR[GP1:90,1] + 14.476;
   1:  PR[GP1:91,2] = PR[GP1:90,2] + 45.110;
   1:L PR[91] R[100]mm/sec CNT100;
   1:  PR[GP1:91,1] = PR[GP1:90,1] + 8.910;
   1:  PR[GP1:91,2] = PR[GP1:90,2] + 45.799;
   1:L PR[91] R[100]mm/sec CNT100;
   1:  PR[GP1:91,1] = PR[GP1:90,1] + 0.594;
   1:  PR[GP1:91,2] = PR[GP1:90,2] + 45.620;
   1:L PR[91] R[100]mm/sec CNT100;
   1:  ! -- Layer/Ebene 187 -- !;
   1:  PR[91] = PR[90];
   1:  PR[GP1:91,1] = PR[GP1:90,1] + -0.361;
   1:  PR[GP1:91,2] = PR[GP1:90,2] + 45.776;
   1:  PR[GP1:91,3] = PR[GP1:90,3] + 114.375;
   1:L PR[91] R[100]mm/sec CNT100;
   1:  PR[GP1:91,1] = PR[GP1:90,1] + -8.327;
   1:  PR[GP1:91,2] = PR[GP1:90,2] + 45.947;
   1:L PR[91] R[100]mm/sec CNT100;
   1:  PR[GP1:91,1] = PR[GP1:90,1] + -14.166;
   1:  PR[GP1:91,2] = PR[GP1:90,2] + 45.224;
   1:L PR[91] R[100]mm/sec CNT100;
   1:  PR[GP1:91,1] = PR[GP1:90,1] + -22.173;
   1:  PR[GP1:91,2] = PR[GP1:90,2] + 42.529;
   1:L PR[91] R[100]mm/sec CNT100;
   1:  PR[GP1:91,1] = PR[GP1:90,1] + -27.368;
   1:  PR[GP1:91,2] = PR[GP1:90,2] + 40.516;
   1:L PR[91] R[100]mm/sec CNT100;
   1:  PR[GP1:91,1] = PR[GP1:90,1] + -34.306;
   1:  PR[GP1:91,2] = PR[GP1:90,2] + 34.972;
   1:L PR[91] R[100]mm/sec CNT100;
   1:  PR[GP1:91,1] = PR[GP1:90,1] + -38.663;
   1:  PR[GP1:91,2] = PR[GP1:90,2] + 31.887;
   1:L PR[91] R[100]mm/sec CNT100;
   1:  PR[GP1:91,1] = PR[GP1:90,1] + -42.460;
   1:  PR[GP1:91,2] = PR[GP1:90,2] + 27.314;
   1:L PR[91] R[100]mm/sec CNT100;
   1:  PR[GP1:91,1] = PR[GP1:90,1] + -47.034;
   1:  PR[GP1:91,2] = PR[GP1:90,2] + 19.673;
   1:L PR[91] R[100]mm/sec CNT100;
   1:  PR[GP1:91,1] = PR[GP1:90,1] + -49.353;
   1:  PR[GP1:91,2] = PR[GP1:90,2] + 14.419;
   1:L PR[91] R[100]mm/sec CNT100;
   1:  PR[GP1:91,1] = PR[GP1:90,1] + -50.978;
   1:  PR[GP1:91,2] = PR[GP1:90,2] + 5.508;
   1:L PR[91] R[100]mm/sec CNT100;
   1:  PR[GP1:91,1] = PR[GP1:90,1] + -51.754;
   1:  PR[GP1:91,2] = PR[GP1:90,2] + -0.059;
   1:L PR[91] R[100]mm/sec CNT100;
   1:  PR[GP1:91,1] = PR[GP1:90,1] + -50.146;
   1:  PR[GP1:91,2] = PR[GP1:90,2] + -8.850;
   1:L PR[91] R[100]mm/sec CNT100;
   1:  PR[GP1:91,1] = PR[GP1:90,1] + -49.348;
   1:  PR[GP1:91,2] = PR[GP1:90,2] + -14.575;
   1:L PR[91] R[100]mm/sec CNT100;
   1:  PR[GP1:91,1] = PR[GP1:90,1] + -47.034;
   1:  PR[GP1:91,2] = PR[GP1:90,2] + -19.816;
   1:L PR[91] R[100]mm/sec CNT100;
   1:  PR[GP1:91,1] = PR[GP1:90,1] + -42.461;
   1:  PR[GP1:91,2] = PR[GP1:90,2] + -27.457;
   1:L PR[91] R[100]mm/sec CNT100;
   1:  PR[GP1:91,1] = PR[GP1:90,1] + -38.652;
   1:  PR[GP1:91,2] = PR[GP1:90,2] + -32.044;
   1:L PR[91] R[100]mm/sec CNT100;
   1:  PR[GP1:91,1] = PR[GP1:90,1] + -31.944;
   1:  PR[GP1:91,2] = PR[GP1:90,2] + -37.425;
   1:L PR[91] R[100]mm/sec CNT100;
   1:  PR[GP1:91,1] = PR[GP1:90,1] + -27.386;
   1:  PR[GP1:91,2] = PR[GP1:90,2] + -40.652;
   1:L PR[91] R[100]mm/sec CNT100;
   1:  PR[GP1:91,1] = PR[GP1:90,1] + -22.174;
   1:  PR[GP1:91,2] = PR[GP1:90,2] + -42.672;
   1:L PR[91] R[100]mm/sec CNT100;
   1:  PR[GP1:91,1] = PR[GP1:90,1] + -14.168;
   1:  PR[GP1:91,2] = PR[GP1:90,2] + -45.367;
   1:L PR[91] R[100]mm/sec CNT100;
   1:  PR[GP1:91,1] = PR[GP1:90,1] + -8.329;
   1:  PR[GP1:91,2] = PR[GP1:90,2] + -46.091;
   1:L PR[91] R[100]mm/sec CNT100;
   1:  PR[GP1:91,1] = PR[GP1:90,1] + -0.362;
   1:  PR[GP1:91,2] = PR[GP1:90,2] + -45.920;
   1:L PR[91] R[100]mm/sec CNT100;
   1:  PR[GP1:91,1] = PR[GP1:90,1] + 0.574;
   1:L PR[91] R[100]mm/sec CNT100;
   1:  PR[GP1:91,1] = PR[GP1:90,1] + 8.542;
   1:  PR[GP1:91,2] = PR[GP1:90,2] + -46.091;
   1:L PR[91] R[100]mm/sec CNT100;
   1:  PR[GP1:91,1] = PR[GP1:90,1] + 14.381;
   1:  PR[GP1:91,2] = PR[GP1:90,2] + -45.368;
   1:L PR[91] R[100]mm/sec CNT100;
   1:  PR[GP1:91,1] = PR[GP1:90,1] + 22.388;
   1:  PR[GP1:91,2] = PR[GP1:90,2] + -42.672;
   1:L PR[91] R[100]mm/sec CNT100;
   1:  PR[GP1:91,1] = PR[GP1:90,1] + 27.584;
   1:  PR[GP1:91,2] = PR[GP1:90,2] + -40.659;
   1:L PR[91] R[100]mm/sec CNT100;
   1:  PR[GP1:91,1] = PR[GP1:90,1] + 34.521;
   1:  PR[GP1:91,2] = PR[GP1:90,2] + -35.114;
   1:L PR[91] R[100]mm/sec CNT100;
   1:  PR[GP1:91,1] = PR[GP1:90,1] + 38.878;
   1:  PR[GP1:91,2] = PR[GP1:90,2] + -32.028;
   1:L PR[91] R[100]mm/sec CNT100;
   1:  PR[GP1:91,1] = PR[GP1:90,1] + 42.675;
   1:  PR[GP1:91,2] = PR[GP1:90,2] + -27.455;
   1:L PR[91] R[100]mm/sec CNT100;
   1:  PR[GP1:91,1] = PR[GP1:90,1] + 47.247;
   1:  PR[GP1:91,2] = PR[GP1:90,2] + -19.819;
   1:L PR[91] R[100]mm/sec CNT100;
   1:  PR[GP1:91,1] = PR[GP1:90,1] + 49.567;
   1:  PR[GP1:91,2] = PR[GP1:90,2] + -14.566;
   1:L PR[91] R[100]mm/sec CNT100;
   1:  PR[GP1:91,1] = PR[GP1:90,1] + 51.191;
   1:  PR[GP1:91,2] = PR[GP1:90,2] + -5.651;
   1:L PR[91] R[100]mm/sec CNT100;
   1:  PR[GP1:91,1] = PR[GP1:90,1] + 51.967;
   1:  PR[GP1:91,2] = PR[GP1:90,2] + -0.085;
   1:L PR[91] R[100]mm/sec CNT100;
   1:  PR[GP1:91,1] = PR[GP1:90,1] + 50.360;
   1:  PR[GP1:91,2] = PR[GP1:90,2] + 8.709;
   1:L PR[91] R[100]mm/sec CNT100;
   1:  PR[GP1:91,1] = PR[GP1:90,1] + 49.561;
   1:  PR[GP1:91,2] = PR[GP1:90,2] + 14.434;
   1:L PR[91] R[100]mm/sec CNT100;
   1:  PR[GP1:91,1] = PR[GP1:90,1] + 47.247;
   1:  PR[GP1:91,2] = PR[GP1:90,2] + 19.675;
   1:L PR[91] R[100]mm/sec CNT100;
   1:  PR[GP1:91,1] = PR[GP1:90,1] + 42.674;
   1:  PR[GP1:91,2] = PR[GP1:90,2] + 27.312;
   1:L PR[91] R[100]mm/sec CNT100;
   1:  PR[GP1:91,1] = PR[GP1:90,1] + 38.866;
   1:  PR[GP1:91,2] = PR[GP1:90,2] + 31.899;
   1:L PR[91] R[100]mm/sec CNT100;
   1:  PR[GP1:91,1] = PR[GP1:90,1] + 32.157;
   1:  PR[GP1:91,2] = PR[GP1:90,2] + 37.281;
   1:L PR[91] R[100]mm/sec CNT100;
   1:  PR[GP1:91,1] = PR[GP1:90,1] + 27.599;
   1:  PR[GP1:91,2] = PR[GP1:90,2] + 40.509;
   1:L PR[91] R[100]mm/sec CNT100;
   1:  PR[GP1:91,1] = PR[GP1:90,1] + 22.386;
   1:  PR[GP1:91,2] = PR[GP1:90,2] + 42.529;
   1:L PR[91] R[100]mm/sec CNT100;
   1:  PR[GP1:91,1] = PR[GP1:90,1] + 14.379;
   1:  PR[GP1:91,2] = PR[GP1:90,2] + 45.224;
   1:L PR[91] R[100]mm/sec CNT100;
   1:  PR[GP1:91,1] = PR[GP1:90,1] + 8.540;
   1:  PR[GP1:91,2] = PR[GP1:90,2] + 45.947;
   1:L PR[91] R[100]mm/sec CNT100;
   1:  PR[GP1:91,1] = PR[GP1:90,1] + 0.573;
   1:  PR[GP1:91,2] = PR[GP1:90,2] + 45.776;
   1:L PR[91] R[100]mm/sec CNT100;
   1:  ! -- Layer/Ebene 188 -- !;
   1:  PR[91] = PR[90];
   1:  PR[GP1:91,1] = PR[GP1:90,1] + -0.341;
   1:  PR[GP1:91,2] = PR[GP1:90,2] + 45.931;
   1:  PR[GP1:91,3] = PR[GP1:90,3] + 114.985;
   1:L PR[91] R[100]mm/sec CNT100;
   1:  PR[GP1:91,1] = PR[GP1:90,1] + -7.956;
   1:  PR[GP1:91,2] = PR[GP1:90,2] + 46.095;
   1:L PR[91] R[100]mm/sec CNT100;
   1:  PR[GP1:91,1] = PR[GP1:90,1] + -14.069;
   1:  PR[GP1:91,2] = PR[GP1:90,2] + 45.338;
   1:L PR[91] R[100]mm/sec CNT100;
   1:  PR[GP1:91,1] = PR[GP1:90,1] + -21.723;
   1:  PR[GP1:91,2] = PR[GP1:90,2] + 42.762;
   1:L PR[91] R[100]mm/sec CNT100;
   1:  PR[GP1:91,1] = PR[GP1:90,1] + -27.188;
   1:  PR[GP1:91,2] = PR[GP1:90,2] + 40.644;
   1:L PR[91] R[100]mm/sec CNT100;
   1:  PR[GP1:91,1] = PR[GP1:90,1] + -33.820;
   1:  PR[GP1:91,2] = PR[GP1:90,2] + 35.345;
   1:L PR[91] R[100]mm/sec CNT100;
   1:  PR[GP1:91,1] = PR[GP1:90,1] + -38.423;
   1:  PR[GP1:91,2] = PR[GP1:90,2] + 32.086;
   1:L PR[91] R[100]mm/sec CNT100;
   1:  PR[GP1:91,1] = PR[GP1:90,1] + -42.436;
   1:  PR[GP1:91,2] = PR[GP1:90,2] + 27.252;
   1:L PR[91] R[100]mm/sec CNT100;
   1:  PR[GP1:91,1] = PR[GP1:90,1] + -46.808;
   1:  PR[GP1:91,2] = PR[GP1:90,2] + 19.949;
   1:L PR[91] R[100]mm/sec CNT100;
   1:  PR[GP1:91,1] = PR[GP1:90,1] + -49.268;
   1:  PR[GP1:91,2] = PR[GP1:90,2] + 14.376;
   1:L PR[91] R[100]mm/sec CNT100;
   1:  PR[GP1:91,1] = PR[GP1:90,1] + -50.821;
   1:  PR[GP1:91,2] = PR[GP1:90,2] + 5.858;
   1:L PR[91] R[100]mm/sec CNT100;
   1:  PR[GP1:91,1] = PR[GP1:90,1] + -51.646;
   1:  PR[GP1:91,2] = PR[GP1:90,2] + -0.059;
   1:L PR[91] R[100]mm/sec CNT100;
   1:  PR[GP1:91,1] = PR[GP1:90,1] + -50.109;
   1:  PR[GP1:91,2] = PR[GP1:90,2] + -8.461;
   1:L PR[91] R[100]mm/sec CNT100;
   1:  PR[GP1:91,1] = PR[GP1:90,1] + -49.263;
   1:  PR[GP1:91,2] = PR[GP1:90,2] + -14.531;
   1:L PR[91] R[100]mm/sec CNT100;
   1:  PR[GP1:91,1] = PR[GP1:90,1] + -46.808;
   1:  PR[GP1:91,2] = PR[GP1:90,2] + -20.092;
   1:L PR[91] R[100]mm/sec CNT100;
   1:  PR[GP1:91,1] = PR[GP1:90,1] + -42.437;
   1:  PR[GP1:91,2] = PR[GP1:90,2] + -27.395;
   1:L PR[91] R[100]mm/sec CNT100;
   1:  PR[GP1:91,1] = PR[GP1:90,1] + -38.412;
   1:  PR[GP1:91,2] = PR[GP1:90,2] + -32.243;
   1:L PR[91] R[100]mm/sec CNT100;
   1:  PR[GP1:91,1] = PR[GP1:90,1] + -32.000;
   1:  PR[GP1:91,2] = PR[GP1:90,2] + -37.386;
   1:L PR[91] R[100]mm/sec CNT100;
   1:  PR[GP1:91,1] = PR[GP1:90,1] + -27.206;
   1:  PR[GP1:91,2] = PR[GP1:90,2] + -40.781;
   1:L PR[91] R[100]mm/sec CNT100;
   1:  PR[GP1:91,1] = PR[GP1:90,1] + -21.724;
   1:  PR[GP1:91,2] = PR[GP1:90,2] + -42.905;
   1:L PR[91] R[100]mm/sec CNT100;
   1:  PR[GP1:91,1] = PR[GP1:90,1] + -14.071;
   1:  PR[GP1:91,2] = PR[GP1:90,2] + -45.482;
   1:L PR[91] R[100]mm/sec CNT100;
   1:  PR[GP1:91,1] = PR[GP1:90,1] + -7.958;
   1:  PR[GP1:91,2] = PR[GP1:90,2] + -46.239;
   1:L PR[91] R[100]mm/sec CNT100;
   1:  PR[GP1:91,1] = PR[GP1:90,1] + -0.342;
   1:  PR[GP1:91,2] = PR[GP1:90,2] + -46.075;
   1:L PR[91] R[100]mm/sec CNT100;
   1:  PR[GP1:91,1] = PR[GP1:90,1] + 0.554;
   1:L PR[91] R[100]mm/sec CNT100;
   1:  PR[GP1:91,1] = PR[GP1:90,1] + 8.171;
   1:  PR[GP1:91,2] = PR[GP1:90,2] + -46.239;
   1:L PR[91] R[100]mm/sec CNT100;
   1:  PR[GP1:91,1] = PR[GP1:90,1] + 14.285;
   1:  PR[GP1:91,2] = PR[GP1:90,2] + -45.482;
   1:L PR[91] R[100]mm/sec CNT100;
   1:  PR[GP1:91,1] = PR[GP1:90,1] + 21.938;
   1:  PR[GP1:91,2] = PR[GP1:90,2] + -42.905;
   1:L PR[91] R[100]mm/sec CNT100;
   1:  PR[GP1:91,1] = PR[GP1:90,1] + 27.403;
   1:  PR[GP1:91,2] = PR[GP1:90,2] + -40.787;
   1:L PR[91] R[100]mm/sec CNT100;
   1:  PR[GP1:91,1] = PR[GP1:90,1] + 34.034;
   1:  PR[GP1:91,2] = PR[GP1:90,2] + -35.487;
   1:L PR[91] R[100]mm/sec CNT100;
   1:  PR[GP1:91,1] = PR[GP1:90,1] + 38.638;
   1:  PR[GP1:91,2] = PR[GP1:90,2] + -32.227;
   1:L PR[91] R[100]mm/sec CNT100;
   1:  PR[GP1:91,1] = PR[GP1:90,1] + 42.651;
   1:  PR[GP1:91,2] = PR[GP1:90,2] + -27.393;
   1:L PR[91] R[100]mm/sec CNT100;
   1:  PR[GP1:91,1] = PR[GP1:90,1] + 47.021;
   1:  PR[GP1:91,2] = PR[GP1:90,2] + -20.094;
   1:L PR[91] R[100]mm/sec CNT100;
   1:  PR[GP1:91,1] = PR[GP1:90,1] + 49.481;
   1:  PR[GP1:91,2] = PR[GP1:90,2] + -14.522;
   1:L PR[91] R[100]mm/sec CNT100;
   1:  PR[GP1:91,1] = PR[GP1:90,1] + 51.034;
   1:  PR[GP1:91,2] = PR[GP1:90,2] + -6.002;
   1:L PR[91] R[100]mm/sec CNT100;
   1:  PR[GP1:91,1] = PR[GP1:90,1] + 51.859;
   1:  PR[GP1:91,2] = PR[GP1:90,2] + -0.085;
   1:L PR[91] R[100]mm/sec CNT100;
   1:  PR[GP1:91,1] = PR[GP1:90,1] + 50.323;
   1:  PR[GP1:91,2] = PR[GP1:90,2] + 8.320;
   1:L PR[91] R[100]mm/sec CNT100;
   1:  PR[GP1:91,1] = PR[GP1:90,1] + 49.476;
   1:  PR[GP1:91,2] = PR[GP1:90,2] + 14.390;
   1:L PR[91] R[100]mm/sec CNT100;
   1:  PR[GP1:91,1] = PR[GP1:90,1] + 47.021;
   1:  PR[GP1:91,2] = PR[GP1:90,2] + 19.951;
   1:L PR[91] R[100]mm/sec CNT100;
   1:  PR[GP1:91,1] = PR[GP1:90,1] + 42.650;
   1:  PR[GP1:91,2] = PR[GP1:90,2] + 27.250;
   1:L PR[91] R[100]mm/sec CNT100;
   1:  PR[GP1:91,1] = PR[GP1:90,1] + 38.626;
   1:  PR[GP1:91,2] = PR[GP1:90,2] + 32.098;
   1:L PR[91] R[100]mm/sec CNT100;
   1:  PR[GP1:91,1] = PR[GP1:90,1] + 32.213;
   1:  PR[GP1:91,2] = PR[GP1:90,2] + 37.242;
   1:L PR[91] R[100]mm/sec CNT100;
   1:  PR[GP1:91,1] = PR[GP1:90,1] + 27.419;
   1:  PR[GP1:91,2] = PR[GP1:90,2] + 40.638;
   1:L PR[91] R[100]mm/sec CNT100;
   1:  PR[GP1:91,1] = PR[GP1:90,1] + 21.936;
   1:  PR[GP1:91,2] = PR[GP1:90,2] + 42.762;
   1:L PR[91] R[100]mm/sec CNT100;
   1:  PR[GP1:91,1] = PR[GP1:90,1] + 14.283;
   1:  PR[GP1:91,2] = PR[GP1:90,2] + 45.338;
   1:L PR[91] R[100]mm/sec CNT100;
   1:  PR[GP1:91,1] = PR[GP1:90,1] + 8.169;
   1:  PR[GP1:91,2] = PR[GP1:90,2] + 46.095;
   1:L PR[91] R[100]mm/sec CNT100;
   1:  PR[GP1:91,1] = PR[GP1:90,1] + 0.553;
   1:  PR[GP1:91,2] = PR[GP1:90,2] + 45.931;
   1:L PR[91] R[100]mm/sec CNT100;
   1:  ! -- Layer/Ebene 189 -- !;
   1:  PR[91] = PR[90];
   1:  PR[GP1:91,1] = PR[GP1:90,1] + -0.321;
   1:  PR[GP1:91,2] = PR[GP1:90,2] + 46.087;
   1:  PR[GP1:91,3] = PR[GP1:90,3] + 115.595;
   1:L PR[91] R[100]mm/sec CNT100;
   1:  PR[GP1:91,1] = PR[GP1:90,1] + -7.586;
   1:  PR[GP1:91,2] = PR[GP1:90,2] + 46.243;
   1:L PR[91] R[100]mm/sec CNT100;
   1:  PR[GP1:91,1] = PR[GP1:90,1] + -13.973;
   1:  PR[GP1:91,2] = PR[GP1:90,2] + 45.452;
   1:L PR[91] R[100]mm/sec CNT100;
   1:  PR[GP1:91,1] = PR[GP1:90,1] + -21.272;
   1:  PR[GP1:91,2] = PR[GP1:90,2] + 42.995;
   1:L PR[91] R[100]mm/sec CNT100;
   1:  PR[GP1:91,1] = PR[GP1:90,1] + -27.008;
   1:  PR[GP1:91,2] = PR[GP1:90,2] + 40.773;
   1:L PR[91] R[100]mm/sec CNT100;
   1:  PR[GP1:91,1] = PR[GP1:90,1] + -33.333;
   1:  PR[GP1:91,2] = PR[GP1:90,2] + 35.719;
   1:L PR[91] R[100]mm/sec CNT100;
   1:  PR[GP1:91,1] = PR[GP1:90,1] + -38.182;
   1:  PR[GP1:91,2] = PR[GP1:90,2] + 32.285;
   1:L PR[91] R[100]mm/sec CNT100;
   1:  PR[GP1:91,1] = PR[GP1:90,1] + -42.412;
   1:  PR[GP1:91,2] = PR[GP1:90,2] + 27.190;
   1:L PR[91] R[100]mm/sec CNT100;
   1:  PR[GP1:91,1] = PR[GP1:90,1] + -46.582;
   1:  PR[GP1:91,2] = PR[GP1:90,2] + 20.224;
   1:L PR[91] R[100]mm/sec CNT100;
   1:  PR[GP1:91,1] = PR[GP1:90,1] + -49.183;
   1:  PR[GP1:91,2] = PR[GP1:90,2] + 14.333;
   1:L PR[91] R[100]mm/sec CNT100;
   1:  PR[GP1:91,1] = PR[GP1:90,1] + -50.664;
   1:  PR[GP1:91,2] = PR[GP1:90,2] + 6.209;
   1:L PR[91] R[100]mm/sec CNT100;
   1:  PR[GP1:91,1] = PR[GP1:90,1] + -51.538;
   1:  PR[GP1:91,2] = PR[GP1:90,2] + -0.059;
   1:L PR[91] R[100]mm/sec CNT100;
   1:  PR[GP1:91,1] = PR[GP1:90,1] + -50.072;
   1:  PR[GP1:91,2] = PR[GP1:90,2] + -8.072;
   1:L PR[91] R[100]mm/sec CNT100;
   1:  PR[GP1:91,1] = PR[GP1:90,1] + -49.178;
   1:  PR[GP1:91,2] = PR[GP1:90,2] + -14.488;
   1:L PR[91] R[100]mm/sec CNT100;
   1:  PR[GP1:91,1] = PR[GP1:90,1] + -46.582;
   1:  PR[GP1:91,2] = PR[GP1:90,2] + -20.368;
   1:L PR[91] R[100]mm/sec CNT100;
   1:  PR[GP1:91,1] = PR[GP1:90,1] + -42.413;
   1:  PR[GP1:91,2] = PR[GP1:90,2] + -27.333;
   1:L PR[91] R[100]mm/sec CNT100;
   1:  PR[GP1:91,1] = PR[GP1:90,1] + -38.171;
   1:  PR[GP1:91,2] = PR[GP1:90,2] + -32.442;
   1:L PR[91] R[100]mm/sec CNT100;
   1:  PR[GP1:91,1] = PR[GP1:90,1] + -32.056;
   1:  PR[GP1:91,2] = PR[GP1:90,2] + -37.347;
   1:L PR[91] R[100]mm/sec CNT100;
   1:  PR[GP1:91,1] = PR[GP1:90,1] + -27.025;
   1:  PR[GP1:91,2] = PR[GP1:90,2] + -40.909;
   1:L PR[91] R[100]mm/sec CNT100;
   1:  PR[GP1:91,1] = PR[GP1:90,1] + -21.274;
   1:  PR[GP1:91,2] = PR[GP1:90,2] + -43.138;
   1:L PR[91] R[100]mm/sec CNT100;
   1:  PR[GP1:91,1] = PR[GP1:90,1] + -13.975;
   1:  PR[GP1:91,2] = PR[GP1:90,2] + -45.596;
   1:L PR[91] R[100]mm/sec CNT100;
   1:  PR[GP1:91,1] = PR[GP1:90,1] + -7.588;
   1:  PR[GP1:91,2] = PR[GP1:90,2] + -46.387;
   1:L PR[91] R[100]mm/sec CNT100;
   1:  PR[GP1:91,1] = PR[GP1:90,1] + -0.321;
   1:  PR[GP1:91,2] = PR[GP1:90,2] + -46.231;
   1:L PR[91] R[100]mm/sec CNT100;
   1:  PR[GP1:91,1] = PR[GP1:90,1] + 0.533;
   1:L PR[91] R[100]mm/sec CNT100;
   1:  PR[GP1:91,1] = PR[GP1:90,1] + 7.800;
   1:  PR[GP1:91,2] = PR[GP1:90,2] + -46.387;
   1:L PR[91] R[100]mm/sec CNT100;
   1:  PR[GP1:91,1] = PR[GP1:90,1] + 14.188;
   1:  PR[GP1:91,2] = PR[GP1:90,2] + -45.596;
   1:L PR[91] R[100]mm/sec CNT100;
   1:  PR[GP1:91,1] = PR[GP1:90,1] + 21.487;
   1:  PR[GP1:91,2] = PR[GP1:90,2] + -43.138;
   1:L PR[91] R[100]mm/sec CNT100;
   1:  PR[GP1:91,1] = PR[GP1:90,1] + 27.223;
   1:  PR[GP1:91,2] = PR[GP1:90,2] + -40.916;
   1:L PR[91] R[100]mm/sec CNT100;
   1:  PR[GP1:91,1] = PR[GP1:90,1] + 33.547;
   1:  PR[GP1:91,2] = PR[GP1:90,2] + -35.860;
   1:L PR[91] R[100]mm/sec CNT100;
   1:  PR[GP1:91,1] = PR[GP1:90,1] + 38.398;
   1:  PR[GP1:91,2] = PR[GP1:90,2] + -32.426;
   1:L PR[91] R[100]mm/sec CNT100;
   1:  PR[GP1:91,1] = PR[GP1:90,1] + 42.627;
   1:  PR[GP1:91,2] = PR[GP1:90,2] + -27.331;
   1:L PR[91] R[100]mm/sec CNT100;
   1:  PR[GP1:91,1] = PR[GP1:90,1] + 46.795;
   1:  PR[GP1:91,2] = PR[GP1:90,2] + -20.370;
   1:L PR[91] R[100]mm/sec CNT100;
   1:  PR[GP1:91,1] = PR[GP1:90,1] + 49.396;
   1:  PR[GP1:91,2] = PR[GP1:90,2] + -14.479;
   1:L PR[91] R[100]mm/sec CNT100;
   1:  PR[GP1:91,1] = PR[GP1:90,1] + 50.877;
   1:  PR[GP1:91,2] = PR[GP1:90,2] + -6.353;
   1:L PR[91] R[100]mm/sec CNT100;
   1:  PR[GP1:91,1] = PR[GP1:90,1] + 51.751;
   1:  PR[GP1:91,2] = PR[GP1:90,2] + -0.085;
   1:L PR[91] R[100]mm/sec CNT100;
   1:  PR[GP1:91,1] = PR[GP1:90,1] + 50.286;
   1:  PR[GP1:91,2] = PR[GP1:90,2] + 7.932;
   1:L PR[91] R[100]mm/sec CNT100;
   1:  PR[GP1:91,1] = PR[GP1:90,1] + 49.391;
   1:  PR[GP1:91,2] = PR[GP1:90,2] + 14.347;
   1:L PR[91] R[100]mm/sec CNT100;
   1:  PR[GP1:91,1] = PR[GP1:90,1] + 46.795;
   1:  PR[GP1:91,2] = PR[GP1:90,2] + 20.226;
   1:L PR[91] R[100]mm/sec CNT100;
   1:  PR[GP1:91,1] = PR[GP1:90,1] + 42.626;
   1:  PR[GP1:91,2] = PR[GP1:90,2] + 27.188;
   1:L PR[91] R[100]mm/sec CNT100;
   1:  PR[GP1:91,1] = PR[GP1:90,1] + 38.385;
   1:  PR[GP1:91,2] = PR[GP1:90,2] + 32.297;
   1:L PR[91] R[100]mm/sec CNT100;
   1:  PR[GP1:91,1] = PR[GP1:90,1] + 32.269;
   1:  PR[GP1:91,2] = PR[GP1:90,2] + 37.203;
   1:L PR[91] R[100]mm/sec CNT100;
   1:  PR[GP1:91,1] = PR[GP1:90,1] + 27.238;
   1:  PR[GP1:91,2] = PR[GP1:90,2] + 40.766;
   1:L PR[91] R[100]mm/sec CNT100;
   1:  PR[GP1:91,1] = PR[GP1:90,1] + 21.486;
   1:  PR[GP1:91,2] = PR[GP1:90,2] + 42.995;
   1:L PR[91] R[100]mm/sec CNT100;
   1:  PR[GP1:91,1] = PR[GP1:90,1] + 14.186;
   1:  PR[GP1:91,2] = PR[GP1:90,2] + 45.452;
   1:L PR[91] R[100]mm/sec CNT100;
   1:  PR[GP1:91,1] = PR[GP1:90,1] + 7.798;
   1:  PR[GP1:91,2] = PR[GP1:90,2] + 46.243;
   1:L PR[91] R[100]mm/sec CNT100;
   1:  PR[GP1:91,1] = PR[GP1:90,1] + 0.533;
   1:  PR[GP1:91,2] = PR[GP1:90,2] + 46.087;
   1:L PR[91] R[100]mm/sec CNT100;
   1:  ! -- Layer/Ebene 190 -- !;
   1:  PR[91] = PR[90];
   1:  PR[GP1:91,1] = PR[GP1:90,1] + -0.301;
   1:  PR[GP1:91,2] = PR[GP1:90,2] + 46.242;
   1:  PR[GP1:91,3] = PR[GP1:90,3] + 116.205;
   1:L PR[91] R[100]mm/sec CNT100;
   1:  PR[GP1:91,1] = PR[GP1:90,1] + -7.215;
   1:  PR[GP1:91,2] = PR[GP1:90,2] + 46.391;
   1:L PR[91] R[100]mm/sec CNT100;
   1:  PR[GP1:91,1] = PR[GP1:90,1] + -13.876;
   1:  PR[GP1:91,2] = PR[GP1:90,2] + 45.566;
   1:L PR[91] R[100]mm/sec CNT100;
   1:  PR[GP1:91,1] = PR[GP1:90,1] + -20.822;
   1:  PR[GP1:91,2] = PR[GP1:90,2] + 43.228;
   1:L PR[91] R[100]mm/sec CNT100;
   1:  PR[GP1:91,1] = PR[GP1:90,1] + -26.827;
   1:  PR[GP1:91,2] = PR[GP1:90,2] + 40.901;
   1:L PR[91] R[100]mm/sec CNT100;
   1:  PR[GP1:91,1] = PR[GP1:90,1] + -32.846;
   1:  PR[GP1:91,2] = PR[GP1:90,2] + 36.092;
   1:L PR[91] R[100]mm/sec CNT100;
   1:  PR[GP1:91,1] = PR[GP1:90,1] + -37.942;
   1:  PR[GP1:91,2] = PR[GP1:90,2] + 32.484;
   1:L PR[91] R[100]mm/sec CNT100;
   1:  PR[GP1:91,1] = PR[GP1:90,1] + -42.388;
   1:  PR[GP1:91,2] = PR[GP1:90,2] + 27.128;
   1:L PR[91] R[100]mm/sec CNT100;
   1:  PR[GP1:91,1] = PR[GP1:90,1] + -46.356;
   1:  PR[GP1:91,2] = PR[GP1:90,2] + 20.500;
   1:L PR[91] R[100]mm/sec CNT100;
   1:  PR[GP1:91,1] = PR[GP1:90,1] + -49.097;
   1:  PR[GP1:91,2] = PR[GP1:90,2] + 14.290;
   1:L PR[91] R[100]mm/sec CNT100;
   1:  PR[GP1:91,1] = PR[GP1:90,1] + -50.507;
   1:  PR[GP1:91,2] = PR[GP1:90,2] + 6.560;
   1:L PR[91] R[100]mm/sec CNT100;
   1:  PR[GP1:91,1] = PR[GP1:90,1] + -51.430;
   1:  PR[GP1:91,2] = PR[GP1:90,2] + -0.059;
   1:L PR[91] R[100]mm/sec CNT100;
   1:  PR[GP1:91,1] = PR[GP1:90,1] + -50.035;
   1:  PR[GP1:91,2] = PR[GP1:90,2] + -7.684;
   1:L PR[91] R[100]mm/sec CNT100;
   1:  PR[GP1:91,1] = PR[GP1:90,1] + -49.092;
   1:  PR[GP1:91,2] = PR[GP1:90,2] + -14.445;
   1:L PR[91] R[100]mm/sec CNT100;
   1:  PR[GP1:91,1] = PR[GP1:90,1] + -46.356;
   1:  PR[GP1:91,2] = PR[GP1:90,2] + -20.644;
   1:L PR[91] R[100]mm/sec CNT100;
   1:  PR[GP1:91,1] = PR[GP1:90,1] + -42.389;
   1:  PR[GP1:91,2] = PR[GP1:90,2] + -27.271;
   1:L PR[91] R[100]mm/sec CNT100;
   1:  PR[GP1:91,1] = PR[GP1:90,1] + -37.931;
   1:  PR[GP1:91,2] = PR[GP1:90,2] + -32.641;
   1:L PR[91] R[100]mm/sec CNT100;
   1:  PR[GP1:91,1] = PR[GP1:90,1] + -32.112;
   1:  PR[GP1:91,2] = PR[GP1:90,2] + -37.308;
   1:L PR[91] R[100]mm/sec CNT100;
   1:  PR[GP1:91,1] = PR[GP1:90,1] + -26.845;
   1:  PR[GP1:91,2] = PR[GP1:90,2] + -41.038;
   1:L PR[91] R[100]mm/sec CNT100;
   1:  PR[GP1:91,1] = PR[GP1:90,1] + -20.823;
   1:  PR[GP1:91,2] = PR[GP1:90,2] + -43.372;
   1:L PR[91] R[100]mm/sec CNT100;
   1:  PR[GP1:91,1] = PR[GP1:90,1] + -13.878;
   1:  PR[GP1:91,2] = PR[GP1:90,2] + -45.710;
   1:L PR[91] R[100]mm/sec CNT100;
   1:  PR[GP1:91,1] = PR[GP1:90,1] + -7.217;
   1:  PR[GP1:91,2] = PR[GP1:90,2] + -46.535;
   1:L PR[91] R[100]mm/sec CNT100;
   1:  PR[GP1:91,1] = PR[GP1:90,1] + -0.301;
   1:  PR[GP1:91,2] = PR[GP1:90,2] + -46.386;
   1:L PR[91] R[100]mm/sec CNT100;
   1:  PR[GP1:91,1] = PR[GP1:90,1] + 0.513;
   1:L PR[91] R[100]mm/sec CNT100;
   1:  PR[GP1:91,1] = PR[GP1:90,1] + 7.429;
   1:  PR[GP1:91,2] = PR[GP1:90,2] + -46.535;
   1:L PR[91] R[100]mm/sec CNT100;
   1:  PR[GP1:91,1] = PR[GP1:90,1] + 14.091;
   1:  PR[GP1:91,2] = PR[GP1:90,2] + -45.710;
   1:L PR[91] R[100]mm/sec CNT100;
   1:  PR[GP1:91,1] = PR[GP1:90,1] + 21.037;
   1:  PR[GP1:91,2] = PR[GP1:90,2] + -43.372;
   1:L PR[91] R[100]mm/sec CNT100;
   1:  PR[GP1:91,1] = PR[GP1:90,1] + 27.042;
   1:  PR[GP1:91,2] = PR[GP1:90,2] + -41.044;
   1:L PR[91] R[100]mm/sec CNT100;
   1:  PR[GP1:91,1] = PR[GP1:90,1] + 33.061;
   1:  PR[GP1:91,2] = PR[GP1:90,2] + -36.234;
   1:L PR[91] R[100]mm/sec CNT100;
   1:  PR[GP1:91,1] = PR[GP1:90,1] + 38.157;
   1:  PR[GP1:91,2] = PR[GP1:90,2] + -32.625;
   1:L PR[91] R[100]mm/sec CNT100;
   1:  PR[GP1:91,1] = PR[GP1:90,1] + 42.603;
   1:  PR[GP1:91,2] = PR[GP1:90,2] + -27.269;
   1:L PR[91] R[100]mm/sec CNT100;
   1:  PR[GP1:91,1] = PR[GP1:90,1] + 46.569;
   1:  PR[GP1:91,2] = PR[GP1:90,2] + -20.646;
   1:L PR[91] R[100]mm/sec CNT100;
   1:  PR[GP1:91,1] = PR[GP1:90,1] + 49.311;
   1:  PR[GP1:91,2] = PR[GP1:90,2] + -14.436;
   1:L PR[91] R[100]mm/sec CNT100;
   1:  PR[GP1:91,1] = PR[GP1:90,1] + 50.720;
   1:  PR[GP1:91,2] = PR[GP1:90,2] + -6.703;
   1:L PR[91] R[100]mm/sec CNT100;
   1:  PR[GP1:91,1] = PR[GP1:90,1] + 51.643;
   1:  PR[GP1:91,2] = PR[GP1:90,2] + -0.085;
   1:L PR[91] R[100]mm/sec CNT100;
   1:  PR[GP1:91,1] = PR[GP1:90,1] + 50.249;
   1:  PR[GP1:91,2] = PR[GP1:90,2] + 7.543;
   1:L PR[91] R[100]mm/sec CNT100;
   1:  PR[GP1:91,1] = PR[GP1:90,1] + 49.306;
   1:  PR[GP1:91,2] = PR[GP1:90,2] + 14.304;
   1:L PR[91] R[100]mm/sec CNT100;
   1:  PR[GP1:91,1] = PR[GP1:90,1] + 46.569;
   1:  PR[GP1:91,2] = PR[GP1:90,2] + 20.502;
   1:L PR[91] R[100]mm/sec CNT100;
   1:  PR[GP1:91,1] = PR[GP1:90,1] + 42.602;
   1:  PR[GP1:91,2] = PR[GP1:90,2] + 27.126;
   1:L PR[91] R[100]mm/sec CNT100;
   1:  PR[GP1:91,1] = PR[GP1:90,1] + 38.145;
   1:  PR[GP1:91,2] = PR[GP1:90,2] + 32.496;
   1:L PR[91] R[100]mm/sec CNT100;
   1:  PR[GP1:91,1] = PR[GP1:90,1] + 32.325;
   1:  PR[GP1:91,2] = PR[GP1:90,2] + 37.164;
   1:L PR[91] R[100]mm/sec CNT100;
   1:  PR[GP1:91,1] = PR[GP1:90,1] + 27.058;
   1:  PR[GP1:91,2] = PR[GP1:90,2] + 40.895;
   1:L PR[91] R[100]mm/sec CNT100;
   1:  PR[GP1:91,1] = PR[GP1:90,1] + 21.035;
   1:  PR[GP1:91,2] = PR[GP1:90,2] + 43.228;
   1:L PR[91] R[100]mm/sec CNT100;
   1:  PR[GP1:91,1] = PR[GP1:90,1] + 14.089;
   1:  PR[GP1:91,2] = PR[GP1:90,2] + 45.566;
   1:L PR[91] R[100]mm/sec CNT100;
   1:  PR[GP1:91,1] = PR[GP1:90,1] + 7.428;
   1:  PR[GP1:91,2] = PR[GP1:90,2] + 46.391;
   1:L PR[91] R[100]mm/sec CNT100;
   1:  PR[GP1:91,1] = PR[GP1:90,1] + 0.513;
   1:  PR[GP1:91,2] = PR[GP1:90,2] + 46.242;
   1:L PR[91] R[100]mm/sec CNT100;
   1:  ! -- Layer/Ebene 191 -- !;
   1:  PR[91] = PR[90];
   1:  PR[GP1:91,1] = PR[GP1:90,1] + -0.281;
   1:  PR[GP1:91,2] = PR[GP1:90,2] + 46.398;
   1:  PR[GP1:91,3] = PR[GP1:90,3] + 116.815;
   1:L PR[91] R[100]mm/sec CNT100;
   1:  PR[GP1:91,1] = PR[GP1:90,1] + -6.845;
   1:  PR[GP1:91,2] = PR[GP1:90,2] + 46.539;
   1:L PR[91] R[100]mm/sec CNT100;
   1:  PR[GP1:91,1] = PR[GP1:90,1] + -13.779;
   1:  PR[GP1:91,2] = PR[GP1:90,2] + 45.680;
   1:L PR[91] R[100]mm/sec CNT100;
   1:  PR[GP1:91,1] = PR[GP1:90,1] + -20.372;
   1:  PR[GP1:91,2] = PR[GP1:90,2] + 43.461;
   1:L PR[91] R[100]mm/sec CNT100;
   1:  PR[GP1:91,1] = PR[GP1:90,1] + -26.647;
   1:  PR[GP1:91,2] = PR[GP1:90,2] + 41.030;
   1:L PR[91] R[100]mm/sec CNT100;
   1:  PR[GP1:91,1] = PR[GP1:90,1] + -32.360;
   1:  PR[GP1:91,2] = PR[GP1:90,2] + 36.465;
   1:L PR[91] R[100]mm/sec CNT100;
   1:  PR[GP1:91,1] = PR[GP1:90,1] + -37.701;
   1:  PR[GP1:91,2] = PR[GP1:90,2] + 32.683;
   1:L PR[91] R[100]mm/sec CNT100;
   1:  PR[GP1:91,1] = PR[GP1:90,1] + -42.365;
   1:  PR[GP1:91,2] = PR[GP1:90,2] + 27.066;
   1:L PR[91] R[100]mm/sec CNT100;
   1:  PR[GP1:91,1] = PR[GP1:90,1] + -46.130;
   1:  PR[GP1:91,2] = PR[GP1:90,2] + 20.776;
   1:L PR[91] R[100]mm/sec CNT100;
   1:  PR[GP1:91,1] = PR[GP1:90,1] + -49.012;
   1:  PR[GP1:91,2] = PR[GP1:90,2] + 14.247;
   1:L PR[91] R[100]mm/sec CNT100;
   1:  PR[GP1:91,1] = PR[GP1:90,1] + -50.350;
   1:  PR[GP1:91,2] = PR[GP1:90,2] + 6.910;
   1:L PR[91] R[100]mm/sec CNT100;
   1:  PR[GP1:91,1] = PR[GP1:90,1] + -51.322;
   1:  PR[GP1:91,2] = PR[GP1:90,2] + -0.059;
   1:L PR[91] R[100]mm/sec CNT100;
   1:  PR[GP1:91,1] = PR[GP1:90,1] + -49.998;
   1:  PR[GP1:91,2] = PR[GP1:90,2] + -7.295;
   1:L PR[91] R[100]mm/sec CNT100;
   1:  PR[GP1:91,1] = PR[GP1:90,1] + -49.007;
   1:  PR[GP1:91,2] = PR[GP1:90,2] + -14.402;
   1:L PR[91] R[100]mm/sec CNT100;
   1:  PR[GP1:91,1] = PR[GP1:90,1] + -46.130;
   1:  PR[GP1:91,2] = PR[GP1:90,2] + -20.919;
   1:L PR[91] R[100]mm/sec CNT100;
   1:  PR[GP1:91,1] = PR[GP1:90,1] + -42.365;
   1:  PR[GP1:91,2] = PR[GP1:90,2] + -27.209;
   1:L PR[91] R[100]mm/sec CNT100;
   1:  PR[GP1:91,1] = PR[GP1:90,1] + -37.690;
   1:  PR[GP1:91,2] = PR[GP1:90,2] + -32.840;
   1:L PR[91] R[100]mm/sec CNT100;
   1:  PR[GP1:91,1] = PR[GP1:90,1] + -32.168;
   1:  PR[GP1:91,2] = PR[GP1:90,2] + -37.269;
   1:L PR[91] R[100]mm/sec CNT100;
   1:  PR[GP1:91,1] = PR[GP1:90,1] + -26.665;
   1:  PR[GP1:91,2] = PR[GP1:90,2] + -41.166;
   1:L PR[91] R[100]mm/sec CNT100;
   1:  PR[GP1:91,1] = PR[GP1:90,1] + -20.373;
   1:  PR[GP1:91,2] = PR[GP1:90,2] + -43.605;
   1:L PR[91] R[100]mm/sec CNT100;
   1:  PR[GP1:91,1] = PR[GP1:90,1] + -13.781;
   1:  PR[GP1:91,2] = PR[GP1:90,2] + -45.824;
   1:L PR[91] R[100]mm/sec CNT100;
   1:  PR[GP1:91,1] = PR[GP1:90,1] + -6.846;
   1:  PR[GP1:91,2] = PR[GP1:90,2] + -46.683;
   1:L PR[91] R[100]mm/sec CNT100;
   1:  PR[GP1:91,1] = PR[GP1:90,1] + -0.281;
   1:  PR[GP1:91,2] = PR[GP1:90,2] + -46.542;
   1:L PR[91] R[100]mm/sec CNT100;
   1:  PR[GP1:91,1] = PR[GP1:90,1] + 0.493;
   1:L PR[91] R[100]mm/sec CNT100;
   1:  PR[GP1:91,1] = PR[GP1:90,1] + 7.059;
   1:  PR[GP1:91,2] = PR[GP1:90,2] + -46.683;
   1:L PR[91] R[100]mm/sec CNT100;
   1:  PR[GP1:91,1] = PR[GP1:90,1] + 13.994;
   1:  PR[GP1:91,2] = PR[GP1:90,2] + -45.824;
   1:L PR[91] R[100]mm/sec CNT100;
   1:  PR[GP1:91,1] = PR[GP1:90,1] + 20.586;
   1:  PR[GP1:91,2] = PR[GP1:90,2] + -43.605;
   1:L PR[91] R[100]mm/sec CNT100;
   1:  PR[GP1:91,1] = PR[GP1:90,1] + 26.862;
   1:  PR[GP1:91,2] = PR[GP1:90,2] + -41.173;
   1:L PR[91] R[100]mm/sec CNT100;
   1:  PR[GP1:91,1] = PR[GP1:90,1] + 32.574;
   1:  PR[GP1:91,2] = PR[GP1:90,2] + -36.607;
   1:L PR[91] R[100]mm/sec CNT100;
   1:  PR[GP1:91,1] = PR[GP1:90,1] + 37.917;
   1:  PR[GP1:91,2] = PR[GP1:90,2] + -32.824;
   1:L PR[91] R[100]mm/sec CNT100;
   1:  PR[GP1:91,1] = PR[GP1:90,1] + 42.579;
   1:  PR[GP1:91,2] = PR[GP1:90,2] + -27.207;
   1:L PR[91] R[100]mm/sec CNT100;
   1:  PR[GP1:91,1] = PR[GP1:90,1] + 46.343;
   1:  PR[GP1:91,2] = PR[GP1:90,2] + -20.921;
   1:L PR[91] R[100]mm/sec CNT100;
   1:  PR[GP1:91,1] = PR[GP1:90,1] + 49.226;
   1:  PR[GP1:91,2] = PR[GP1:90,2] + -14.392;
   1:L PR[91] R[100]mm/sec CNT100;
   1:  PR[GP1:91,1] = PR[GP1:90,1] + 50.563;
   1:  PR[GP1:91,2] = PR[GP1:90,2] + -7.054;
   1:L PR[91] R[100]mm/sec CNT100;
   1:  PR[GP1:91,1] = PR[GP1:90,1] + 51.535;
   1:  PR[GP1:91,2] = PR[GP1:90,2] + -0.085;
   1:L PR[91] R[100]mm/sec CNT100;
   1:  PR[GP1:91,1] = PR[GP1:90,1] + 50.212;
   1:  PR[GP1:91,2] = PR[GP1:90,2] + 7.154;
   1:L PR[91] R[100]mm/sec CNT100;
   1:  PR[GP1:91,1] = PR[GP1:90,1] + 49.220;
   1:  PR[GP1:91,2] = PR[GP1:90,2] + 14.260;
   1:L PR[91] R[100]mm/sec CNT100;
   1:  PR[GP1:91,1] = PR[GP1:90,1] + 46.343;
   1:  PR[GP1:91,2] = PR[GP1:90,2] + 20.778;
   1:L PR[91] R[100]mm/sec CNT100;
   1:  PR[GP1:91,1] = PR[GP1:90,1] + 42.578;
   1:  PR[GP1:91,2] = PR[GP1:90,2] + 27.064;
   1:L PR[91] R[100]mm/sec CNT100;
   1:  PR[GP1:91,1] = PR[GP1:90,1] + 37.904;
   1:  PR[GP1:91,2] = PR[GP1:90,2] + 32.695;
   1:L PR[91] R[100]mm/sec CNT100;
   1:  PR[GP1:91,1] = PR[GP1:90,1] + 32.382;
   1:  PR[GP1:91,2] = PR[GP1:90,2] + 37.125;
   1:L PR[91] R[100]mm/sec CNT100;
   1:  PR[GP1:91,1] = PR[GP1:90,1] + 26.877;
   1:  PR[GP1:91,2] = PR[GP1:90,2] + 41.023;
   1:L PR[91] R[100]mm/sec CNT100;
   1:  PR[GP1:91,1] = PR[GP1:90,1] + 20.585;
   1:  PR[GP1:91,2] = PR[GP1:90,2] + 43.461;
   1:L PR[91] R[100]mm/sec CNT100;
   1:  PR[GP1:91,1] = PR[GP1:90,1] + 13.993;
   1:  PR[GP1:91,2] = PR[GP1:90,2] + 45.680;
   1:L PR[91] R[100]mm/sec CNT100;
   1:  PR[GP1:91,1] = PR[GP1:90,1] + 7.057;
   1:  PR[GP1:91,2] = PR[GP1:90,2] + 46.539;
   1:L PR[91] R[100]mm/sec CNT100;
   1:  PR[GP1:91,1] = PR[GP1:90,1] + 0.492;
   1:  PR[GP1:91,2] = PR[GP1:90,2] + 46.398;
   1:L PR[91] R[100]mm/sec CNT100;
   1:  ! -- Layer/Ebene 192 -- !;
   1:  PR[91] = PR[90];
   1:  PR[GP1:91,1] = PR[GP1:90,1] + -0.261;
   1:  PR[GP1:91,2] = PR[GP1:90,2] + 46.553;
   1:  PR[GP1:91,3] = PR[GP1:90,3] + 117.425;
   1:L PR[91] R[100]mm/sec CNT100;
   1:  PR[GP1:91,1] = PR[GP1:90,1] + -6.474;
   1:  PR[GP1:91,2] = PR[GP1:90,2] + 46.687;
   1:L PR[91] R[100]mm/sec CNT100;
   1:  PR[GP1:91,1] = PR[GP1:90,1] + -13.683;
   1:  PR[GP1:91,2] = PR[GP1:90,2] + 45.794;
   1:L PR[91] R[100]mm/sec CNT100;
   1:  PR[GP1:91,1] = PR[GP1:90,1] + -19.922;
   1:  PR[GP1:91,2] = PR[GP1:90,2] + 43.695;
   1:L PR[91] R[100]mm/sec CNT100;
   1:  PR[GP1:91,1] = PR[GP1:90,1] + -26.467;
   1:  PR[GP1:91,2] = PR[GP1:90,2] + 41.158;
   1:L PR[91] R[100]mm/sec CNT100;
   1:  PR[GP1:91,1] = PR[GP1:90,1] + -31.873;
